	LOCAL CONST Robtarget Tr_meulage_bavure_P130 :=[[66.91934375,115.7860078125,16],[0.0375790299429137,-0.0384114691049443,-0.713777108740491,0.698308395043204],[0,0,0,0],[8.999999E+09,8.999999E+09,8.999999E+09,8.999999E+09,8.999999E+09,8.999999E+09]];
	LOCAL CONST Robtarget Tr_meulage_bavure_P131 :=[[72.78634375,115.0686953125,16],[0.040217072512141,-0.0409917261667762,-0.712641457174476,0.699174097761538],[0,0,0,0],[8.999999E+09,8.999999E+09,8.999999E+09,8.999999E+09,8.999999E+09,8.999999E+09]];
	LOCAL CONST Robtarget Tr_meulage_bavure_P132 :=[[73.607359375,114.957515625,16],[0.0430704475740681,-0.0437750469990952,-0.711474851088136,0.700023012532524],[0,0,0,0],[8.999999E+09,8.999999E+09,8.999999E+09,8.999999E+09,8.999999E+09,8.999999E+09]];
	LOCAL CONST Robtarget Tr_meulage_bavure_P133 :=[[80.8797578125,113.9724765625,16],[0.0463242339768427,-0.0469486652254147,-0.710274730272182,0.70082786454078],[0,0,0,0],[8.999999E+09,8.999999E+09,8.999999E+09,8.999999E+09,8.999999E+09,8.999999E+09]];
	LOCAL CONST Robtarget Tr_meulage_bavure_P134 :=[[81.893921875,113.8622109375,16],[0.0500455236008215,-0.0505782090053766,-0.70903845529879,0.701570922465316],[0,0,0,0],[8.999999E+09,8.999999E+09,8.999999E+09,8.999999E+09,8.999999E+09,8.999999E+09]];
	LOCAL CONST Robtarget Tr_meulage_bavure_P135 :=[[86.0903046875,113.1481953125,16],[0.0541087782813907,-0.0545356720476456,-0.70778179785277,0.702241430859436],[0,0,0,0],[8.999999E+09,8.999999E+09,8.999999E+09,8.999999E+09,8.999999E+09,8.999999E+09]];
	LOCAL CONST Robtarget Tr_meulage_bavure_P136 :=[[87.9428125,112.849546875,16],[0.0582007586477647,-0.0585060712323081,-0.706535976535859,0.70284893482334],[0,0,0,0],[8.999999E+09,8.999999E+09,8.999999E+09,8.999999E+09,8.999999E+09,8.999999E+09]];
	LOCAL CONST Robtarget Tr_meulage_bavure_P137 :=[[89.760375,112.5874921875,16],[0.0619449334526603,-0.0621148803561433,-0.705345034592479,0.703415203868684],[0,0,0,0],[8.999999E+09,8.999999E+09,8.999999E+09,8.999999E+09,8.999999E+09,8.999999E+09]];
	LOCAL CONST Robtarget Tr_meulage_bavure_P138 :=[[96.0940234375,111.0590546875,16],[0.0650697780701425,-0.065095955864691,-0.704246851452174,0.703963644467287],[0,0,0,0],[8.999999E+09,8.999999E+09,8.999999E+09,8.999999E+09,8.999999E+09,8.999999E+09]];
	LOCAL CONST Robtarget Tr_meulage_bavure_P139 :=[[96.4307578125,110.9958203125,16],[0.0675357884502958,-0.0674170712414185,-0.703260439151439,0.704498836413625],[0,0,0,0],[8.999999E+09,8.999999E+09,8.999999E+09,8.999999E+09,8.999999E+09,8.999999E+09]];
	LOCAL CONST Robtarget Tr_meulage_bavure_P140 :=[[106.677734375,109.285953125,16],[0.0695409234803893,-0.0692837834926727,-0.702387001473537,0.704993842148603],[0,0,0,0],[8.999999E+09,8.999999E+09,8.999999E+09,8.999999E+09,8.999999E+09,8.999999E+09]];
	LOCAL CONST Robtarget Tr_meulage_bavure_P141 :=[[106.9891640625,109.2307109375,16],[0.0713921073001013,-0.0710053649896085,-0.70159983106773,0.705421209068508],[0,0,0,0],[8.999999E+09,8.999999E+09,8.999999E+09,8.999999E+09,8.999999E+09,8.999999E+09]];
	LOCAL CONST Robtarget Tr_meulage_bavure_P142 :=[[107.1989453125,109.1865234375,16],[0.0732993553122748,-0.0727933096486914,-0.700883234161866,0.705755645143557],[0,0,0,0],[8.999999E+09,8.999999E+09,8.999999E+09,8.999999E+09,8.999999E+09,8.999999E+09]];
	LOCAL CONST Robtarget Tr_meulage_bavure_P143 :=[[110.56125,108.47396875,16],[0.0752309363699142,-0.0746187293208283,-0.700247555166698,0.705992714502433],[0,0,0,0],[8.999999E+09,8.999999E+09,8.999999E+09,8.999999E+09,8.999999E+09,8.999999E+09]];
	LOCAL CONST Robtarget Tr_meulage_bavure_P144 :=[[111.3198828125,108.289640625,16],[0.0769389781355609,-0.076236764322119,-0.699716860698982,0.706161924959644],[0,0,0,0],[8.999999E+09,8.999999E+09,8.999999E+09,8.999999E+09,8.999999E+09,8.999999E+09]];
	LOCAL CONST Robtarget Tr_meulage_bavure_P145 :=[[112.3602265625,108.048890625,16],[0.0781115130178079,-0.0773402560327233,-0.699326258671287,0.706300120532116],[0,0,0,0],[8.999999E+09,8.999999E+09,8.999999E+09,8.999999E+09,8.999999E+09,8.999999E+09]];
	LOCAL CONST Robtarget Tr_meulage_bavure_P146 :=[[114.5588359375,107.543515625,16],[0.0785747149746875,-0.0777587433548293,-0.699095336504751,0.706431385539907],[0,0,0,0],[8.999999E+09,8.999999E+09,8.999999E+09,8.999999E+09,8.999999E+09,8.999999E+09]];
	LOCAL CONST Robtarget Tr_meulage_bavure_P147 :=[[115.668765625,107.266140625,16],[0.0784214795360947,-0.0775843590394273,-0.699009918050557,0.706552102287415],[0,0,0,0],[8.999999E+09,8.999999E+09,8.999999E+09,8.999999E+09,8.999999E+09,8.999999E+09]];
	LOCAL CONST Robtarget Tr_meulage_bavure_P148 :=[[117.5694609375,106.84359375,16],[0.0780069203121761,-0.0771676079432631,-0.699025386011006,0.706628325486524],[0,0,0,0],[8.999999E+09,8.999999E+09,8.999999E+09,8.999999E+09,8.999999E+09,8.999999E+09]];
	LOCAL CONST Robtarget Tr_meulage_bavure_P149 :=[[118.382015625,106.655640625,16],[0.0777860523380435,-0.0769565613223954,-0.699083246410587,0.706618448895251],[0,0,0,0],[8.999999E+09,8.999999E+09,8.999999E+09,8.999999E+09,8.999999E+09,8.999999E+09]];
	LOCAL CONST Robtarget Tr_meulage_bavure_P150 :=[[121.6917734375,105.9990546875,16],[0.0781312083527598,-0.077318092245178,-0.699136115354537,0.706488583842563],[0,0,0,0],[8.999999E+09,8.999999E+09,8.999999E+09,8.999999E+09,8.999999E+09,8.999999E+09]];
	LOCAL CONST Robtarget Tr_meulage_bavure_P151 :=[[125.2111171875,105.2392265625,16],[0.0792169084017852,-0.078423438108987,-0.699154110679908,0.706227991018351],[0,0,0,0],[8.999999E+09,8.999999E+09,8.999999E+09,8.999999E+09,8.999999E+09,8.999999E+09]];
	LOCAL CONST Robtarget Tr_meulage_bavure_P152 :=[[126.6580234375,104.8870234375,16],[0.0809905250458525,-0.0802193534282553,-0.699128968723034,0.705849895714816],[0,0,0,0],[8.999999E+09,8.999999E+09,8.999999E+09,8.999999E+09,8.999999E+09,8.999999E+09]];
	LOCAL CONST Robtarget Tr_meulage_bavure_P153 :=[[129.6603984375,104.143984375,16],[0.0832551345128652,-0.0825101821253249,-0.699069483083656,0.705381109928555],[0,0,0,0],[8.999999E+09,8.999999E+09,8.999999E+09,8.999999E+09,8.999999E+09,8.999999E+09]];
	LOCAL CONST Robtarget Tr_meulage_bavure_P154 :=[[136.354125,102.4169609375,16],[0.0857848622766101,-0.0850709210273251,-0.698988120213109,0.70485424280534],[0,0,0,0],[8.999999E+09,8.999999E+09,8.999999E+09,8.999999E+09,8.999999E+09,8.999999E+09]];
	LOCAL CONST Robtarget Tr_meulage_bavure_P155 :=[[137.42846875,102.1511875,16],[0.0884091672402083,-0.0877319052022491,-0.698897826468415,0.704293092480114],[0,0,0,0],[8.999999E+09,8.999999E+09,8.999999E+09,8.999999E+09,8.999999E+09,8.999999E+09]];
	LOCAL CONST Robtarget Tr_meulage_bavure_P156 :=[[144.5833125,100.26434375,16],[0.0910431915599839,-0.0904067032944326,-0.698798168569051,0.703717901487908],[0,0,0,0],[8.999999E+09,8.999999E+09,8.999999E+09,8.999999E+09,8.999999E+09,8.999999E+09]];
	LOCAL CONST Robtarget Tr_meulage_bavure_P157 :=[[146.926640625,99.6148046875,16],[0.0936691483507536,-0.0930756350342028,-0.698683585512406,0.703138865478046],[0,0,0,0],[8.999999E+09,8.999999E+09,8.999999E+09,8.999999E+09,8.999999E+09,8.999999E+09]];
	LOCAL CONST Robtarget Tr_meulage_bavure_P158 :=[[150.95953125,98.4415625,16],[0.0962879304034066,-0.0957394224747977,-0.69855392139274,0.702556059222072],[0,0,0,0],[8.999999E+09,8.999999E+09,8.999999E+09,8.999999E+09,8.999999E+09,8.999999E+09]];
	LOCAL CONST Robtarget Tr_meulage_bavure_P159 :=[[153.138734375,97.7918125,16],[0.0988916895437435,-0.0983883422839826,-0.698404120332552,0.701977102578359],[0,0,0,0],[8.999999E+09,8.999999E+09,8.999999E+09,8.999999E+09,8.999999E+09,8.999999E+09]];
	LOCAL CONST Robtarget Tr_meulage_bavure_P160 :=[[157.757078125,96.4455546875,16],[0.101440612933847,-0.100981536227335,-0.698236939472659,0.701411225847311],[0,0,0,0],[8.999999E+09,8.999999E+09,8.999999E+09,8.999999E+09,8.999999E+09,8.999999E+09]];
	LOCAL CONST Robtarget Tr_meulage_bavure_P161 :=[[158.63409375,96.21628125,16],[0.103869656310797,-0.103455017724827,-0.698066701122684,0.70086449088902],[0,0,0,0],[8.999999E+09,8.999999E+09,8.999999E+09,8.999999E+09,8.999999E+09,8.999999E+09]];
	LOCAL CONST Robtarget Tr_meulage_bavure_P162 :=[[161.731328125,95.3334375,16],[0.106127055185058,-0.105757019641076,-0.697903326027202,0.700345235205147],[0,0,0,0],[8.999999E+09,8.999999E+09,8.999999E+09,8.999999E+09,8.999999E+09,8.999999E+09]];
	LOCAL CONST Robtarget Tr_meulage_bavure_P163 :=[[163.41271875,94.773984375,16],[0.108205069351474,-0.107879192972837,-0.697749227537857,0.699856955499119],[0,0,0,0],[8.999999E+09,8.999999E+09,8.999999E+09,8.999999E+09,8.999999E+09,8.999999E+09]];
	LOCAL CONST Robtarget Tr_meulage_bavure_P164 :=[[168.711796875,93.117984375,16],[0.110163902620429,-0.109882603679943,-0.697601214294859,0.699387070070852],[0,0,0,0],[8.999999E+09,8.999999E+09,8.999999E+09,8.999999E+09,8.999999E+09,8.999999E+09]];
	LOCAL CONST Robtarget Tr_meulage_bavure_P165 :=[[169.002984375,93.037046875,16],[0.112115837692814,-0.11188027121235,-0.697446164040501,0.698914652956339],[0,0,0,0],[8.999999E+09,8.999999E+09,8.999999E+09,8.999999E+09,8.999999E+09,8.999999E+09]];
	LOCAL CONST Robtarget Tr_meulage_bavure_P166 :=[[175.044734375,91.0927421875,16],[0.114161085801191,-0.113974890865321,-0.697275818516395,0.698414922272729],[0,0,0,0],[8.999999E+09,8.999999E+09,8.999999E+09,8.999999E+09,8.999999E+09,8.999999E+09]];
	LOCAL CONST Robtarget Tr_meulage_bavure_P167 :=[[175.713875,90.8525703125,16],[0.116327655332839,-0.116195967636685,-0.697088341701476,0.697878368753198],[0,0,0,0],[8.999999E+09,8.999999E+09,8.999999E+09,8.999999E+09,8.999999E+09,8.999999E+09]];
	LOCAL CONST Robtarget Tr_meulage_bavure_P168 :=[[177.1794375,90.3878515625,16],[0.118529478570234,-0.118459490986501,-0.696901735552245,0.697313475195594],[0,0,0,0],[8.999999E+09,8.999999E+09,8.999999E+09,8.999999E+09,8.999999E+09,8.999999E+09]];
	LOCAL CONST Robtarget Tr_meulage_bavure_P169 :=[[180.194765625,89.338625,16],[0.120588784077744,-0.120590468458572,-0.696753129059677,0.69674339696702],[0,0,0,0],[8.999999E+09,8.999999E+09,8.999999E+09,8.999999E+09,8.999999E+09,8.999999E+09]];
	LOCAL CONST Robtarget Tr_meulage_bavure_P170 :=[[182.01146875,88.6708671875,16],[0.122306368602409,-0.122391776429605,-0.696684495612379,0.696198332973458],[0,0,0,0],[8.999999E+09,8.999999E+09,8.999999E+09,8.999999E+09,8.999999E+09,8.999999E+09]];
	LOCAL CONST Robtarget Tr_meulage_bavure_P171 :=[[185.929625,87.2135,16],[0.123567193506988,-0.123751009683332,-0.696727295823529,0.695692397217042],[0,0,0,0],[8.999999E+09,8.999999E+09,8.999999E+09,8.999999E+09,8.999999E+09,8.999999E+09]];
	LOCAL CONST Robtarget Tr_meulage_bavure_P172 :=[[187.18065625,86.7315078125,16],[0.124415620474812,-0.124713739181367,-0.696880996836631,0.695215155825341],[0,0,0,0],[8.999999E+09,8.999999E+09,8.999999E+09,8.999999E+09,8.999999E+09,8.999999E+09]];
	LOCAL CONST Robtarget Tr_meulage_bavure_P173 :=[[189.04584375,86.04696875,16],[0.125074969784971,-0.125504974941815,-0.697111566398052,0.69472312268428],[0,0,0,0],[8.999999E+09,8.999999E+09,8.999999E+09,8.999999E+09,8.999999E+09,8.999999E+09]];
	LOCAL CONST Robtarget Tr_meulage_bavure_P174 :=[[190.664125,85.3816796875,16],[0.125898358033854,-0.126480701100316,-0.697359329420033,0.694148544163563],[0,0,0,0],[8.999999E+09,8.999999E+09,8.999999E+09,8.999999E+09,8.999999E+09,8.999999E+09]];
	LOCAL CONST Robtarget Tr_meulage_bavure_P175 :=[[192.474609375,84.74475,16],[0.127251837277854,-0.128012368352486,-0.697561606568862,0.693417340783504],[0,0,0,0],[8.999999E+09,8.999999E+09,8.999999E+09,8.999999E+09,8.999999E+09,8.999999E+09]];
	LOCAL CONST Robtarget Tr_meulage_bavure_P176 :=[[194.93378125,83.8551015625,16],[0.129383618966927,-0.130354980774212,-0.697672769672953,0.692473945060207],[0,0,0,0],[8.999999E+09,8.999999E+09,8.999999E+09,8.999999E+09,8.999999E+09,8.999999E+09]];
	LOCAL CONST Robtarget Tr_meulage_bavure_P177 :=[[196.478875,83.225859375,16],[0.132323925738124,-0.133543900842516,-0.697677993470186,0.691304435579891],[0,0,0,0],[8.999999E+09,8.999999E+09,8.999999E+09,8.999999E+09,8.999999E+09,8.999999E+09]];
	LOCAL CONST Robtarget Tr_meulage_bavure_P178 :=[[200.12365625,81.8095390625,16],[0.135877207452713,-0.137388271043078,-0.697605868715162,0.689933257213197],[0,0,0,0],[8.999999E+09,8.999999E+09,8.999999E+09,8.999999E+09,8.999999E+09,8.999999E+09]];
	LOCAL CONST Robtarget Tr_meulage_bavure_P179 :=[[202.561578125,80.75653125,16],[0.139685278222459,-0.141531070512551,-0.697518656155899,0.688421893494065],[0,0,0,0],[8.999999E+09,8.999999E+09,8.999999E+09,8.999999E+09,8.999999E+09,8.999999E+09]];
	LOCAL CONST Robtarget Tr_meulage_bavure_P180 :=[[207.698796875,78.43090625,16],[0.143350747480375,-0.145574635078128,-0.697498867206909,0.686843445818453],[0,0,0,0],[8.999999E+09,8.999999E+09,8.999999E+09,8.999999E+09,8.999999E+09,8.999999E+09]];
	LOCAL CONST Robtarget Tr_meulage_bavure_P181 :=[[209.555171875,77.6030546875,16],[0.146540725641296,-0.149180855171853,-0.697618889464421,0.685272772873069],[0,0,0,0],[8.999999E+09,8.999999E+09,8.999999E+09,8.999999E+09,8.999999E+09,8.999999E+09]];
	LOCAL CONST Robtarget Tr_meulage_bavure_P182 :=[[210.891359375,77.0095234375,16],[0.149040228183799,-0.152126413175283,-0.697928299674523,0.68376944455772],[0,0,0,0],[8.999999E+09,8.999999E+09,8.999999E+09,8.999999E+09,8.999999E+09,8.999999E+09]];
	LOCAL CONST Robtarget Tr_meulage_bavure_P183 :=[[212.986875,76.031890625,16],[0.150734443360395,-0.154289349959885,-0.698460976711582,0.682368073758504],[0,0,0,0],[8.999999E+09,8.999999E+09,8.999999E+09,8.999999E+09,8.999999E+09,8.999999E+09]];
	LOCAL CONST Robtarget Tr_meulage_bavure_P184 :=[[217.078546875,74.016234375,16],[0.151570317945741,-0.155607772630321,-0.699233612155391,0.681091047839407],[0,0,0,0],[8.999999E+09,8.999999E+09,8.999999E+09,8.999999E+09,8.999999E+09,8.999999E+09]];
	LOCAL CONST Robtarget Tr_meulage_bavure_P185 :=[[218.941953125,73.112125,16],[0.151569402372408,-0.156092119138138,-0.700237370211066,0.679948227416857],[0,0,0,0],[8.999999E+09,8.999999E+09,8.999999E+09,8.999999E+09,8.999999E+09,8.999999E+09]];
	LOCAL CONST Robtarget Tr_meulage_bavure_P186 :=[[219.0621875,73.06121875,16],[0.150837702259073,-0.155840185661068,-0.701442332980961,0.678925973588103],[0,0,0,0],[8.999999E+09,8.999999E+09,8.999999E+09,8.999999E+09,8.999999E+09,8.999999E+09]];
	LOCAL CONST Robtarget Tr_meulage_bavure_P187 :=[[219.1090625,73.033109375,16],[0.149636648993526,-0.155109844533247,-0.702776618858019,0.677978490361863],[0,0,0,0],[8.999999E+09,8.999999E+09,8.999999E+09,8.999999E+09,8.999999E+09,8.999999E+09]];
	LOCAL CONST Robtarget Tr_meulage_bavure_P188 :=[[222.09015625,71.6129140625,16],[0.148574336094181,-0.154522304802513,-0.704087568238217,0.676985391441416],[0,0,0,0],[8.999999E+09,8.999999E+09,8.999999E+09,8.999999E+09,8.999999E+09,8.999999E+09]];
	LOCAL CONST Robtarget Tr_meulage_bavure_P189 :=[[229.641546875,68.055234375,16],[0.148626996287793,-0.155089341077337,-0.705134905379677,0.675752970747344],[0,0,0,0],[8.999999E+09,8.999999E+09,8.999999E+09,8.999999E+09,8.999999E+09,8.999999E+09]];
	LOCAL CONST Robtarget Tr_meulage_bavure_P190 :=[[230.11071875,67.8279140625,16],[0.151271074807113,-0.158361042480802,-0.705554971353023,0.673966634597091],[0,0,0,0],[8.999999E+09,8.999999E+09,8.999999E+09,8.999999E+09,8.999999E+09,8.999999E+09]];
	LOCAL CONST Robtarget Tr_meulage_bavure_P191 :=[[233.1743125,66.54559375,16],[0.158480102126182,-0.166430569449805,-0.704809140639182,0.671140073348438],[0,0,0,0],[8.999999E+09,8.999999E+09,8.999999E+09,8.999999E+09,8.999999E+09,8.999999E+09]];
	LOCAL CONST Robtarget Tr_meulage_bavure_P192 :=[[233.944765625,66.22134375,16],[0.172471661081484,-0.181663624911472,-0.702094674614285,0.666569517294393],[0,0,0,0],[8.999999E+09,8.999999E+09,8.999999E+09,8.999999E+09,8.999999E+09,8.999999E+09]];
	LOCAL CONST Robtarget Tr_meulage_bavure_P193 :=[[234.4685,65.9126875,16],[0.195272456379888,-0.206245163845634,-0.696254711205549,0.659212391641518],[0,0,0,0],[8.999999E+09,8.999999E+09,8.999999E+09,8.999999E+09,8.999999E+09,8.999999E+09]];
	LOCAL CONST Robtarget Tr_meulage_bavure_P194 :=[[235.857546875,65.32159375,16],[0.227792969698998,-0.24119253559603,-0.685838349962404,0.647736274612836],[0,0,0,0],[8.999999E+09,8.999999E+09,8.999999E+09,8.999999E+09,8.999999E+09,8.999999E+09]];
	LOCAL CONST Robtarget Tr_meulage_bavure_P195 :=[[237.085015625,64.44748046875,16],[0.268887533298227,-0.285326947579369,-0.669496083625712,0.63092235768886],[0,0,0,0],[8.999999E+09,8.999999E+09,8.999999E+09,8.999999E+09,8.999999E+09,8.999999E+09]];
	LOCAL CONST Robtarget Tr_meulage_bavure_P196 :=[[237.9425625,63.1903984375,16],[0.314996141790336,-0.334870453464709,-0.646850326102626,0.608460241654678],[0,0,0,0],[8.999999E+09,8.999999E+09,8.999999E+09,8.999999E+09,8.999999E+09,8.999999E+09]];
	LOCAL CONST Robtarget Tr_meulage_bavure_P197 :=[[238.0418125,63.07073828125,16],[0.361424808772667,-0.384786321985673,-0.619044160812946,0.581460162848475],[0,0,0,0],[8.999999E+09,8.999999E+09,8.999999E+09,8.999999E+09,8.999999E+09,8.999999E+09]];
	LOCAL CONST Robtarget Tr_meulage_bavure_P198 :=[[238.087640625,62.9619765625,16],[0.404605659191079,-0.431207701831069,-0.588094753981249,0.551814043652256],[0,0,0,0],[8.999999E+09,8.999999E+09,8.999999E+09,8.999999E+09,8.999999E+09,8.999999E+09]];
	LOCAL CONST Robtarget Tr_meulage_bavure_P199 :=[[238.506046875,60.62127734375,16],[0.443062387855305,-0.472484667298788,-0.555752974041069,0.521145460960772],[0,0,0,0],[8.999999E+09,8.999999E+09,8.999999E+09,8.999999E+09,8.999999E+09,8.999999E+09]];
	LOCAL CONST Robtarget Tr_meulage_bavure_P200 :=[[238.6093125,59.7001328125,16],[0.476650321376658,-0.508389052787827,-0.52319014626542,0.490527382505598],[0,0,0,0],[8.999999E+09,8.999999E+09,8.999999E+09,8.999999E+09,8.999999E+09,8.999999E+09]];
	LOCAL CONST Robtarget Tr_meulage_bavure_P201 :=[[237.7109375,57.469390625,16],[0.505451156136112,-0.53895486429405,-0.491501652997141,0.460947836653485],[0,0,0,0],[8.999999E+09,8.999999E+09,8.999999E+09,8.999999E+09,8.999999E+09,8.999999E+09]];
	LOCAL CONST Robtarget Tr_meulage_bavure_P202 :=[[236.879703125,55.57473828125,16],[0.529331236729187,-0.564002254730795,-0.462148127760641,0.433738407901194],[0,0,0,0],[8.999999E+09,8.999999E+09,8.999999E+09,8.999999E+09,8.999999E+09,8.999999E+09]];
	LOCAL CONST Robtarget Tr_meulage_bavure_P203 :=[[236.66284375,55.11083984375,16],[0.548233372494373,-0.583447016687868,-0.436664316627856,0.410309666697484],[0,0,0,0],[8.999999E+09,8.999999E+09,8.999999E+09,8.999999E+09,8.999999E+09,8.999999E+09]];
	LOCAL CONST Robtarget Tr_meulage_bavure_P204 :=[[235.0753125,52.03003125,16],[0.562452491386192,-0.597603777768636,-0.416104904645074,0.391629452493596],[0,0,0,0],[8.999999E+09,8.999999E+09,8.999999E+09,8.999999E+09,8.999999E+09,8.999999E+09]];
	LOCAL CONST Robtarget Tr_meulage_bavure_P205 :=[[232.848875,47.99112109375,16],[0.572670247409118,-0.607197499281822,-0.400686686586718,0.377902320435371],[0,0,0,0],[8.999999E+09,8.999999E+09,8.999999E+09,8.999999E+09,8.999999E+09,8.999999E+09]];
	LOCAL CONST Robtarget Tr_meulage_bavure_P206 :=[[231.788703125,45.97287109375,16],[0.579797402910104,-0.613235537289396,-0.3898050973045,0.368550042056046],[0,0,0,0],[8.999999E+09,8.999999E+09,8.999999E+09,8.999999E+09,8.999999E+09,8.999999E+09]];
	LOCAL CONST Robtarget Tr_meulage_bavure_P207 :=[[231.750421875,46.01022265625,16],[0.584743800948948,-0.616698687680699,-0.382440881141462,0.362624307371171],[0,0,0,0],[8.999999E+09,8.999999E+09,8.999999E+09,8.999999E+09,8.999999E+09,8.999999E+09]];
	LOCAL CONST Robtarget Tr_meulage_bavure_P208 :=[[230.563046875,43.4813828125,16],[0.588303582827908,-0.618443461707875,-0.377476158934893,0.359079835883867],[0,0,0,0],[8.999999E+09,8.999999E+09,8.999999E+09,8.999999E+09,8.999999E+09,8.999999E+09]];
	LOCAL CONST Robtarget Tr_meulage_bavure_P209 :=[[228.135625,38.742125,16],[0.591075423099639,-0.619138479944678,-0.373956669203322,0.357006717608694],[0,0,0,0],[8.999999E+09,8.999999E+09,8.999999E+09,8.999999E+09,8.999999E+09,8.999999E+09]];
	LOCAL CONST Robtarget Tr_meulage_bavure_P210 :=[[227.6539375,37.97744921875,16],[0.59346983022117,-0.619233588321481,-0.371194119980086,0.355750262127757],[0,0,0,0],[8.999999E+09,8.999999E+09,8.999999E+09,8.999999E+09,8.999999E+09,8.999999E+09]];
	LOCAL CONST Robtarget Tr_meulage_bavure_P211 :=[[227.583375,37.84625390625,16],[0.59578771747521,-0.619083199083303,-0.368651892343638,0.354779890340359],[0,0,0,0],[8.999999E+09,8.999999E+09,8.999999E+09,8.999999E+09,8.999999E+09,8.999999E+09]];
	LOCAL CONST Robtarget Tr_meulage_bavure_P212 :=[[223.232234375,29.75045703125,16],[0.59826322315855,-0.618948699501958,-0.365912211100707,0.353683300380678],[0,0,0,0],[8.999999E+09,8.999999E+09,8.999999E+09,8.999999E+09,8.999999E+09,8.999999E+09]];
	LOCAL CONST Robtarget Tr_meulage_bavure_P213 :=[[222.742609375,28.879546875,16],[0.601110196290616,-0.619074471589474,-0.362582673927974,0.35206126612979],[0,0,0,0],[8.999999E+09,8.999999E+09,8.999999E+09,8.999999E+09,8.999999E+09,8.999999E+09]];
	LOCAL CONST Robtarget Tr_meulage_bavure_P214 :=[[219.652765625,22.688568359375,16],[0.604470518421326,-0.619625642008761,-0.358389216634608,0.349623548298331],[0,0,0,0],[8.999999E+09,8.999999E+09,8.999999E+09,8.999999E+09,8.999999E+09,8.999999E+09]];
	LOCAL CONST Robtarget Tr_meulage_bavure_P215 :=[[218.990046875,21.3121328125,16],[0.608276493688391,-0.620552871503657,-0.353416807429074,0.346425173914026],[0,0,0,0],[8.999999E+09,8.999999E+09,8.999999E+09,8.999999E+09,8.999999E+09,8.999999E+09]];
	LOCAL CONST Robtarget Tr_meulage_bavure_P216 :=[[218.1641875,19.516814453125,16],[0.612202390644332,-0.6215539324952,-0.348209714398515,0.342970751941944],[0,0,0,0],[8.999999E+09,8.999999E+09,8.999999E+09,8.999999E+09,8.999999E+09,8.999999E+09]];
	LOCAL CONST Robtarget Tr_meulage_bavure_P217 :=[[215.843265625,15.1568603515625,16],[0.615711006556747,-0.622118377345017,-0.343722099195397,0.340182009370264],[0,0,0,0],[8.999999E+09,8.999999E+09,8.999999E+09,8.999999E+09,8.999999E+09,8.999999E+09]];
	LOCAL CONST Robtarget Tr_meulage_bavure_P218 :=[[215.603765625,14.73193359375,16],[0.618247194410525,-0.621700174240876,-0.34098922432466,0.339095338875138],[0,0,0,0],[8.999999E+09,8.999999E+09,8.999999E+09,8.999999E+09,8.999999E+09,8.999999E+09]];
	LOCAL CONST Robtarget Tr_meulage_bavure_P219 :=[[215.48725,14.5715634765625,16],[0.619428558964651,-0.619963866268426,-0.340700330946559,0.340406153518684],[0,0,0,0],[8.999999E+09,8.999999E+09,8.999999E+09,8.999999E+09,8.999999E+09,8.999999E+09]];
	LOCAL CONST Robtarget Tr_meulage_bavure_P220 :=[[212.94371875,10.92562890625,16],[0.619189685973086,-0.616882730457898,-0.34291302665433,0.34419541803767],[0,0,0,0],[8.999999E+09,8.999999E+09,8.999999E+09,8.999999E+09,8.999999E+09,8.999999E+09]];
	LOCAL CONST Robtarget Tr_meulage_bavure_P221 :=[[210.711859375,7.6824033203125,16],[0.617793467753272,-0.612757654465243,-0.347038617328745,0.349890677466824],[0,0,0,0],[8.999999E+09,8.999999E+09,8.999999E+09,8.999999E+09,8.999999E+09,8.999999E+09]];
	LOCAL CONST Robtarget Tr_meulage_bavure_P222 :=[[209.336421875,5.25592041015625,16],[0.615729233509894,-0.608088125169878,-0.352115617639173,0.356540228926954],[0,0,0,0],[8.999999E+09,8.999999E+09,8.999999E+09,8.999999E+09,8.999999E+09,8.999999E+09]];
	LOCAL CONST Robtarget Tr_meulage_bavure_P223 :=[[208.604984375,3.98187255859375,16],[0.613532173472829,-0.603419982946631,-0.357177068427192,0.363162688177283],[0,0,0,0],[8.999999E+09,8.999999E+09,8.999999E+09,8.999999E+09,8.999999E+09,8.999999E+09]];
	LOCAL CONST Robtarget Tr_meulage_bavure_P224 :=[[206.372984375,-0.804412841796875,16],[0.611662197159133,-0.59922168111387,-0.361469981964712,0.368974505336019],[0,0,0,0],[8.999999E+09,8.999999E+09,8.999999E+09,8.999999E+09,8.999999E+09,8.999999E+09]];
	LOCAL CONST Robtarget Tr_meulage_bavure_P225 :=[[205.655703125,-2.33804321289063,16],[0.610428440285061,-0.595774575282164,-0.364562330984876,0.373529224513126],[0,0,0,0],[8.999999E+09,8.999999E+09,8.999999E+09,8.999999E+09,8.999999E+09,8.999999E+09]];
	LOCAL CONST Robtarget Tr_meulage_bavure_P226 :=[[205.306515625,-3.13638305664063,16],[0.609970630238294,-0.593221869097205,-0.366292565633338,0.376634306235191],[0,0,0,0],[8.999999E+09,8.999999E+09,8.999999E+09,8.999999E+09,8.999999E+09,8.999999E+09]];
	LOCAL CONST Robtarget Tr_meulage_bavure_P227 :=[[203.0261875,-7.57730078125,16],[0.610287493058713,-0.591562424509279,-0.366711703652052,0.378319441913082],[0,0,0,0],[8.999999E+09,8.999999E+09,8.999999E+09,8.999999E+09,8.999999E+09,8.999999E+09]];
	LOCAL CONST Robtarget Tr_meulage_bavure_P228 :=[[201.42346875,-10.699615234375,16],[0.611273752937712,-0.590676043388691,-0.366019028972191,0.378782630497203],[0,0,0,0],[8.999999E+09,8.999999E+09,8.999999E+09,8.999999E+09,8.999999E+09,8.999999E+09]];
	LOCAL CONST Robtarget Tr_meulage_bavure_P229 :=[[197.501828125,-18.230896484375,16],[0.612750021112551,-0.59039743156596,-0.364498085131601,0.378298070788474],[0,0,0,0],[8.999999E+09,8.999999E+09,8.999999E+09,8.999999E+09,8.999999E+09,8.999999E+09]];
	LOCAL CONST Robtarget Tr_meulage_bavure_P230 :=[[196.443484375,-20.251861328125,16],[0.614519592787454,-0.590532121989523,-0.362455427247399,0.377178401075405],[0,0,0,0],[8.999999E+09,8.999999E+09,8.999999E+09,8.999999E+09,8.999999E+09,8.999999E+09]];
	LOCAL CONST Robtarget Tr_meulage_bavure_P231 :=[[195.890625,-21.320525390625,16],[0.616387866924389,-0.590909198060636,-0.36018303811425,0.375713316520091],[0,0,0,0],[8.999999E+09,8.999999E+09,8.999999E+09,8.999999E+09,8.999999E+09,8.999999E+09]];
	LOCAL CONST Robtarget Tr_meulage_bavure_P232 :=[[192.78528125,-26.824158203125,16],[0.618192759727046,-0.591385952223848,-0.357926574441675,0.374150951678328],[0,0,0,0],[8.999999E+09,8.999999E+09,8.999999E+09,8.999999E+09,8.999999E+09,8.999999E+09]];
	LOCAL CONST Robtarget Tr_meulage_bavure_P233 :=[[191.961296875,-28.487701171875,16],[0.619788398563889,-0.59181878102234,-0.355918672819268,0.372739546833191],[0,0,0,0],[8.999999E+09,8.999999E+09,8.999999E+09,8.999999E+09,8.999999E+09,8.999999E+09]];
	LOCAL CONST Robtarget Tr_meulage_bavure_P234 :=[[191.71503125,-29.23452734375,16],[0.621010587314961,-0.592072467915302,-0.354413234717379,0.371735527272516],[0,0,0,0],[8.999999E+09,8.999999E+09,8.999999E+09,8.999999E+09,8.999999E+09,8.999999E+09]];
	LOCAL CONST Robtarget Tr_meulage_bavure_P235 :=[[191.2190625,-30.219666015625,16],[0.621717150920934,-0.592020916672666,-0.353636981800015,0.371375690610181],[0,0,0,0],[8.999999E+09,8.999999E+09,8.999999E+09,8.999999E+09,8.999999E+09,8.999999E+09]];
	LOCAL CONST Robtarget Tr_meulage_bavure_P236 :=[[190.413390625,-31.797484375,16],[0.621844618805108,-0.591613368888173,-0.35368880301411,0.371762185325999],[0,0,0,0],[8.999999E+09,8.999999E+09,8.999999E+09,8.999999E+09,8.999999E+09,8.999999E+09]];
	LOCAL CONST Robtarget Tr_meulage_bavure_P237 :=[[189.352296875,-33.64605859375,16],[0.621474786784406,-0.590935626905415,-0.354432305698057,0.372749131350752],[0,0,0,0],[8.999999E+09,8.999999E+09,8.999999E+09,8.999999E+09,8.999999E+09,8.999999E+09]];
	LOCAL CONST Robtarget Tr_meulage_bavure_P238 :=[[188.66540625,-34.951109375,16],[0.620853488883399,-0.590218182218205,-0.35547523483033,0.373926196117189],[0,0,0,0],[8.999999E+09,8.999999E+09,8.999999E+09,8.999999E+09,8.999999E+09,8.999999E+09]];
	LOCAL CONST Robtarget Tr_meulage_bavure_P239 :=[[187.039984375,-37.97381640625,16],[0.620336030294727,-0.589817841504478,-0.356247814205903,0.374680688366368],[0,0,0,0],[8.999999E+09,8.999999E+09,8.999999E+09,8.999999E+09,8.999999E+09,8.999999E+09]];
	LOCAL CONST Robtarget Tr_meulage_bavure_P240 :=[[186.095953125,-39.88458203125,16],[0.62027164381349,-0.590046519008715,-0.356213130566664,0.374460143270959],[0,0,0,0],[8.999999E+09,8.999999E+09,8.999999E+09,8.999999E+09,8.999999E+09,8.999999E+09]];
	LOCAL CONST Robtarget Tr_meulage_bavure_P241 :=[[184.659484375,-42.5355234375,16],[0.620848961703628,-0.591075599173121,-0.355073857767026,0.372959459384133],[0,0,0,0],[8.999999E+09,8.999999E+09,8.999999E+09,8.999999E+09,8.999999E+09,8.999999E+09]];
	LOCAL CONST Robtarget Tr_meulage_bavure_P242 :=[[183.497984375,-44.72093359375,16],[0.622007609011476,-0.592853797057783,-0.352903022008749,0.370257162932856],[0,0,0,0],[8.999999E+09,8.999999E+09,8.999999E+09,8.999999E+09,8.999999E+09,8.999999E+09]];
	LOCAL CONST Robtarget Tr_meulage_bavure_P243 :=[[182.948,-45.741546875,16],[0.623470604116682,-0.595107437368185,-0.350120143436793,0.366807073202319],[0,0,0,0],[8.999999E+09,8.999999E+09,8.999999E+09,8.999999E+09,8.999999E+09,8.999999E+09]];
	LOCAL CONST Robtarget Tr_meulage_bavure_P244 :=[[182.502265625,-46.5653671875,16],[0.624830473684378,-0.59744409125455,-0.347369716800421,0.363292880236285],[0,0,0,0],[8.999999E+09,8.999999E+09,8.999999E+09,8.999999E+09,8.999999E+09,8.999999E+09]];
	LOCAL CONST Robtarget Tr_meulage_bavure_P245 :=[[180.579765625,-49.96437109375,16],[0.625689222370143,-0.599454185968829,-0.345326866083021,0.360440052568486],[0,0,0,0],[8.999999E+09,8.999999E+09,8.999999E+09,8.999999E+09,8.999999E+09,8.999999E+09]];
	LOCAL CONST Robtarget Tr_meulage_bavure_P246 :=[[178.879265625,-52.42295703125,16],[0.625787535266007,-0.600881790469465,-0.344450124057943,0.358727120001225],[0,0,0,0],[8.999999E+09,8.999999E+09,8.999999E+09,8.999999E+09,8.999999E+09,8.999999E+09]];
	LOCAL CONST Robtarget Tr_meulage_bavure_P247 :=[[177.75403125,-54.22612109375,16],[0.625096640484182,-0.601683573776541,-0.344817130388136,0.358234858289601],[0,0,0,0],[8.999999E+09,8.999999E+09,8.999999E+09,8.999999E+09,8.999999E+09,8.999999E+09]];
	LOCAL CONST Robtarget Tr_meulage_bavure_P248 :=[[176.502140625,-56.56321875,16],[0.623836157558886,-0.602041809301397,-0.346081948112199,0.358610364554805],[0,0,0,0],[8.999999E+09,8.999999E+09,8.999999E+09,8.999999E+09,8.999999E+09,8.999999E+09]];
	LOCAL CONST Robtarget Tr_meulage_bavure_P249 :=[[174.892328125,-59.35589453125,16],[0.622391120370798,-0.602317688626201,-0.347602406444529,0.359186946151369],[0,0,0,0],[8.999999E+09,8.999999E+09,8.999999E+09,8.999999E+09,8.999999E+09,8.999999E+09]];
	LOCAL CONST Robtarget Tr_meulage_bavure_P250 :=[[174.53259375,-59.8879375,16],[0.621154712377756,-0.602871615478753,-0.348729548041246,0.359305358802084],[0,0,0,0],[8.999999E+09,8.999999E+09,8.999999E+09,8.999999E+09,8.999999E+09,8.999999E+09]];
	LOCAL CONST Robtarget Tr_meulage_bavure_P251 :=[[172.712578125,-63.39216796875,16],[0.620331837491256,-0.603876425402539,-0.349133232445201,0.358646985544475],[0,0,0,0],[8.999999E+09,8.999999E+09,8.999999E+09,8.999999E+09,8.999999E+09,8.999999E+09]];
	LOCAL CONST Robtarget Tr_meulage_bavure_P252 :=[[171.728453125,-65.503203125,16],[0.619805074760416,-0.605222481505007,-0.349003645355567,0.357412748388586],[0,0,0,0],[8.999999E+09,8.999999E+09,8.999999E+09,8.999999E+09,8.999999E+09,8.999999E+09]];
	LOCAL CONST Robtarget Tr_meulage_bavure_P253 :=[[169.82275,-69.12046875,16],[0.619207693908575,-0.60652948670266,-0.348969562751748,0.35626402826764],[0,0,0,0],[8.999999E+09,8.999999E+09,8.999999E+09,8.999999E+09,8.999999E+09,8.999999E+09]];
	LOCAL CONST Robtarget Tr_meulage_bavure_P254 :=[[168.76715625,-71.4039296875,16],[0.618087663420885,-0.607348493401192,-0.349806991606178,0.355992298390918],[0,0,0,0],[8.999999E+09,8.999999E+09,8.999999E+09,8.999999E+09,8.999999E+09,8.999999E+09]];
	LOCAL CONST Robtarget Tr_meulage_bavure_P255 :=[[167.9378125,-73.0588515625,16],[0.616144959830655,-0.607357422873582,-0.352044103976498,0.357137646028848],[0,0,0,0],[8.999999E+09,8.999999E+09,8.999999E+09,8.999999E+09,8.999999E+09,8.999999E+09]];
	LOCAL CONST Robtarget Tr_meulage_bavure_P256 :=[[166.74378125,-75.276609375,16],[0.613378087222688,-0.606536116562397,-0.355676185075052,0.359688355094935],[0,0,0,0],[8.999999E+09,8.999999E+09,8.999999E+09,8.999999E+09,8.999999E+09,8.999999E+09]];
	LOCAL CONST Robtarget Tr_meulage_bavure_P257 :=[[164.823359375,-78.886203125,16],[0.610086762360184,-0.605171452282996,-0.360170676752647,0.363096046993215],[0,0,0,0],[8.999999E+09,8.999999E+09,8.999999E+09,8.999999E+09,8.999999E+09,8.999999E+09]];
	LOCAL CONST Robtarget Tr_meulage_bavure_P258 :=[[164.210265625,-80.159453125,16],[0.6067464359017,-0.603696402987638,-0.364734016579159,0.366576748704014],[0,0,0,0],[8.999999E+09,8.999999E+09,8.999999E+09,8.999999E+09,8.999999E+09,8.999999E+09]];
	LOCAL CONST Robtarget Tr_meulage_bavure_P259 :=[[159.279296875,-90.4268203125,16],[0.603794572049477,-0.602555269633964,-0.368645944214193,0.369404154841761],[0,0,0,0],[8.999999E+09,8.999999E+09,8.999999E+09,8.999999E+09,8.999999E+09,8.999999E+09]];
	LOCAL CONST Robtarget Tr_meulage_bavure_P260 :=[[159.27728125,-90.43153125,16],[0.601509067955308,-0.602016109948271,-0.371480686790883,0.371167810931474],[0,0,0,0],[8.999999E+09,8.999999E+09,8.999999E+09,8.999999E+09,8.999999E+09,8.999999E+09]];
	LOCAL CONST Robtarget Tr_meulage_bavure_P261 :=[[159.273625,-90.4391953125,16],[0.599964120093679,-0.602129628113578,-0.373150575467244,0.371808571144461],[0,0,0,0],[8.999999E+09,8.999999E+09,8.999999E+09,8.999999E+09,8.999999E+09,8.999999E+09]];
	LOCAL CONST Robtarget Tr_meulage_bavure_P262 :=[[158.607421875,-91.55940625,16],[0.599067473064845,-0.602802801286211,-0.373813700067992,0.371497325856694],[0,0,0,0],[8.999999E+09,8.999999E+09,8.999999E+09,8.999999E+09,8.999999E+09,8.999999E+09]];
	LOCAL CONST Robtarget Tr_meulage_bavure_P263 :=[[157.8125625,-93.275375,16],[0.598655714200807,-0.603859956588914,-0.373739036855634,0.370518044113076],[0,0,0,0],[8.999999E+09,8.999999E+09,8.999999E+09,8.999999E+09,8.999999E+09,8.999999E+09]];
	LOCAL CONST Robtarget Tr_meulage_bavure_P264 :=[[156.013921875,-96.855515625,16],[0.598581633581101,-0.605145309120703,-0.373164557711938,0.369117048720652],[0,0,0,0],[8.999999E+09,8.999999E+09,8.999999E+09,8.999999E+09,8.999999E+09,8.999999E+09]];
	LOCAL CONST Robtarget Tr_meulage_bavure_P265 :=[[154.408453125,-99.789203125,16],[0.598741656024643,-0.606547397296493,-0.372258274988102,0.367467632420327],[0,0,0,0],[8.999999E+09,8.999999E+09,8.999999E+09,8.999999E+09,8.999999E+09,8.999999E+09]];
	LOCAL CONST Robtarget Tr_meulage_bavure_P266 :=[[153.829828125,-100.938015625,16],[0.599111908948481,-0.60801253502702,-0.371071109870387,0.365639042261192],[0,0,0,0],[8.999999E+09,8.999999E+09,8.999999E+09,8.999999E+09,8.999999E+09,8.999999E+09]];
	LOCAL CONST Robtarget Tr_meulage_bavure_P267 :=[[153.0649375,-102.244765625,16],[0.599724034156747,-0.609571192908333,-0.369547441468825,0.363577683769115],[0,0,0,0],[8.999999E+09,8.999999E+09,8.999999E+09,8.999999E+09,8.999999E+09,8.999999E+09]];
	LOCAL CONST Robtarget Tr_meulage_bavure_P268 :=[[150.26190625,-107.945859375,16],[0.600618817736741,-0.611240459447048,-0.367626408072759,0.361238094064016],[0,0,0,0],[8.999999E+09,8.999999E+09,8.999999E+09,8.999999E+09,8.999999E+09,8.999999E+09]];
	LOCAL CONST Robtarget Tr_meulage_bavure_P269 :=[[149.97125,-108.5094296875,16],[0.601781252200874,-0.6130081873259,-0.365324582278095,0.358633847195575],[0,0,0,0],[8.999999E+09,8.999999E+09,8.999999E+09,8.999999E+09,8.999999E+09,8.999999E+09]];
	LOCAL CONST Robtarget Tr_meulage_bavure_P270 :=[[149.841921875,-108.737109375,16],[0.603099595811995,-0.614763102362251,-0.362825686515417,0.355942027175726],[0,0,0,0],[8.999999E+09,8.999999E+09,8.999999E+09,8.999999E+09,8.999999E+09,8.999999E+09]];
	LOCAL CONST Robtarget Tr_meulage_bavure_P271 :=[[148.19159375,-111.5269921875,16],[0.604381813712803,-0.616290646069509,-0.360473121939606,0.353507554628702],[0,0,0,0],[8.999999E+09,8.999999E+09,8.999999E+09,8.999999E+09,8.999999E+09,8.999999E+09]];
	LOCAL CONST Robtarget Tr_meulage_bavure_P272 :=[[147.971859375,-111.859875,16],[0.605406221586117,-0.617363609773654,-0.358664431601985,0.351717650531913],[0,0,0,0],[8.999999E+09,8.999999E+09,8.999999E+09,8.999999E+09,8.999999E+09,8.999999E+09]];
	LOCAL CONST Robtarget Tr_meulage_bavure_P273 :=[[147.5519375,-112.6409296875,16],[0.606016266100963,-0.617826031383224,-0.357686791491451,0.350849596492364],[0,0,0,0],[8.999999E+09,8.999999E+09,8.999999E+09,8.999999E+09,8.999999E+09,8.999999E+09]];
	LOCAL CONST Robtarget Tr_meulage_bavure_P274 :=[[146.0570625,-115.0536171875,16],[0.606201132604477,-0.617685600677894,-0.357557374750242,0.35090940327377],[0,0,0,0],[8.999999E+09,8.999999E+09,8.999999E+09,8.999999E+09,8.999999E+09,8.999999E+09]];
	LOCAL CONST Robtarget Tr_meulage_bavure_P275 :=[[143.955203125,-118.973203125,16],[0.606101570923346,-0.617112593766817,-0.358012611863592,0.35162466080361],[0,0,0,0],[8.999999E+09,8.999999E+09,8.999999E+09,8.999999E+09,8.999999E+09,8.999999E+09]];
	LOCAL CONST Robtarget Tr_meulage_bavure_P276 :=[[143.357421875,-120.373765625,16],[0.6059844558601,-0.616377956599261,-0.358581089829075,0.352534616586018],[0,0,0,0],[8.999999E+09,8.999999E+09,8.999999E+09,8.999999E+09,8.999999E+09,8.999999E+09]];
	LOCAL CONST Robtarget Tr_meulage_bavure_P277 :=[[142.211671875,-123.1184375,16],[0.606111846959739,-0.615785572563122,-0.358782110409862,0.353145798287346],[0,0,0,0],[8.999999E+09,8.999999E+09,8.999999E+09,8.999999E+09,8.999999E+09,8.999999E+09]];
	LOCAL CONST Robtarget Tr_meulage_bavure_P278 :=[[141.69628125,-124.1225625,16],[0.606639211689127,-0.615512883122357,-0.358335319481018,0.353169302692116],[0,0,0,0],[8.999999E+09,8.999999E+09,8.999999E+09,8.999999E+09,8.999999E+09,8.999999E+09]];
	LOCAL CONST Robtarget Tr_meulage_bavure_P279 :=[[141.450984375,-124.770234375,16],[0.607551268446271,-0.615555230777337,-0.357261024378716,0.352615618672595],[0,0,0,0],[8.999999E+09,8.999999E+09,8.999999E+09,8.999999E+09,8.999999E+09,8.999999E+09]];
	LOCAL CONST Robtarget Tr_meulage_bavure_P280 :=[[140.48821875,-126.753109375,16],[0.60860471686433,-0.615722965428547,-0.355948085233736,0.351833041473938],[0,0,0,0],[8.999999E+09,8.999999E+09,8.999999E+09,8.999999E+09,8.999999E+09,8.999999E+09]];
	LOCAL CONST Robtarget Tr_meulage_bavure_P281 :=[[139.2965625,-128.884140625,16],[0.609412114607907,-0.615649493857614,-0.355059221578392,0.351461981520233],[0,0,0,0],[8.999999E+09,8.999999E+09,8.999999E+09,8.999999E+09,8.999999E+09,8.999999E+09]];
	LOCAL CONST Robtarget Tr_meulage_bavure_P282 :=[[138.7163125,-129.7308828125,16],[0.609548490329035,-0.61492304981615,-0.355329209696512,0.352223556110109],[0,0,0,0],[8.999999E+09,8.999999E+09,8.999999E+09,8.999999E+09,8.999999E+09,8.999999E+09]];
	LOCAL CONST Robtarget Tr_meulage_bavure_P283 :=[[136.49109375,-133.125578125,16],[0.60869059863804,-0.613253389411855,-0.357287378454986,0.354629052252209],[0,0,0,0],[8.999999E+09,8.999999E+09,8.999999E+09,8.999999E+09,8.999999E+09,8.999999E+09]];
	LOCAL CONST Robtarget Tr_meulage_bavure_P284 :=[[135.589421875,-134.34003125,16],[0.606809153742224,-0.610619816583659,-0.360934203724167,0.358681740700563],[0,0,0,0],[8.999999E+09,8.999999E+09,8.999999E+09,8.999999E+09,8.999999E+09,8.999999E+09]];
	LOCAL CONST Robtarget Tr_meulage_bavure_P285 :=[[134.770875,-135.49840625,16],[0.604187975688785,-0.607362877961505,-0.365692280383206,0.363780676473527],[0,0,0,0],[8.999999E+09,8.999999E+09,8.999999E+09,8.999999E+09,8.999999E+09,8.999999E+09]];
	LOCAL CONST Robtarget Tr_meulage_bavure_P286 :=[[133.573671875,-137.730640625,16],[0.601416707057644,-0.604070711573766,-0.370540372403093,0.368912391104014],[0,0,0,0],[8.999999E+09,8.999999E+09,8.999999E+09,8.999999E+09,8.999999E+09,8.999999E+09]];
	LOCAL CONST Robtarget Tr_meulage_bavure_P287 :=[[133.108828125,-139.018546875,16],[0.599140362240513,-0.601376565025791,-0.374444816355674,0.373052453250817],[0,0,0,0],[8.999999E+09,8.999999E+09,8.999999E+09,8.999999E+09,8.999999E+09,8.999999E+09]];
	LOCAL CONST Robtarget Tr_meulage_bavure_P288 :=[[132.29278125,-140.600125,16],[0.597729431643992,-0.599676521954628,-0.376847655033012,0.375624067997606],[0,0,0,0],[8.999999E+09,8.999999E+09,8.999999E+09,8.999999E+09,8.999999E+09,8.999999E+09]];
	LOCAL CONST Robtarget Tr_meulage_bavure_P289 :=[[131.3254375,-143.260328125,16],[0.597163392446936,-0.598937749449976,-0.377831999251129,0.376712669480281],[0,0,0,0],[8.999999E+09,8.999999E+09,8.999999E+09,8.999999E+09,8.999999E+09,8.999999E+09]];
	LOCAL CONST Robtarget Tr_meulage_bavure_P290 :=[[130.809875,-144.2653125,16],[0.597056893879946,-0.598761785707264,-0.378034432378165,0.376958031329215],[0,0,0,0],[8.999999E+09,8.999999E+09,8.999999E+09,8.999999E+09,8.999999E+09,8.999999E+09]];
	LOCAL CONST Robtarget Tr_meulage_bavure_P291 :=[[130.5497421875,-144.7399375,16],[0.596833034476496,-0.598559817524481,-0.378379007981161,0.377287423752542],[0,0,0,0],[8.999999E+09,8.999999E+09,8.999999E+09,8.999999E+09,8.999999E+09,8.999999E+09]];
	LOCAL CONST Robtarget Tr_meulage_bavure_P292 :=[[130.4254140625,-144.931609375,16],[0.595828133701051,-0.597663354216964,-0.379916045837112,0.378749453111081],[0,0,0,0],[8.999999E+09,8.999999E+09,8.999999E+09,8.999999E+09,8.999999E+09,8.999999E+09]];
	LOCAL CONST Robtarget Tr_meulage_bavure_P293 :=[[126.363828125,-152.60990625,16],[0.593014540964361,-0.595023303575851,-0.384237019461418,0.382939858570397],[0,0,0,0],[8.999999E+09,8.999999E+09,8.999999E+09,8.999999E+09,8.999999E+09,8.999999E+09]];
	LOCAL CONST Robtarget Tr_meulage_bavure_P294 :=[[126.017578125,-153.26628125,16],[0.58537258395462,-0.58758872306254,-0.395763616013899,0.394270961045354],[0,0,0,0],[8.999999E+09,8.999999E+09,8.999999E+09,8.999999E+09,8.999999E+09,8.999999E+09]];
	LOCAL CONST Robtarget Tr_meulage_bavure_P295 :=[[124.9164453125,-155.774171875,16],[0.551261408535918,-0.553617475186278,-0.442312222547626,0.440429845051792],[0,0,0,0],[8.999999E+09,8.999999E+09,8.999999E+09,8.999999E+09,8.999999E+09,8.999999E+09]];
	LOCAL CONST Robtarget Tr_meulage_bavure_P296 :=[[123.527890625,-158.6770625,16],[0.175884491247366,-0.176735690959794,0.686424365405069,-0.683118387878608],[0,0,0,0],[8.999999E+09,8.999999E+09,8.999999E+09,8.999999E+09,8.999999E+09,8.999999E+09]];
	LOCAL CONST Robtarget Tr_meulage_bavure_P297 :=[[123.327640625,-159.0216875,16],[0.306890262185601,-0.308559664737703,0.638359933428414,-0.63490621013334],[0,0,0,0],[8.999999E+09,8.999999E+09,8.999999E+09,8.999999E+09,8.999999E+09,8.999999E+09]];
	LOCAL CONST Robtarget Tr_meulage_bavure_P298 :=[[123.24621875,-159.1608125,16],[0.323837374309504,-0.325798370301669,0.629979367059983,-0.626187491082189],[0,0,0,0],[8.999999E+09,8.999999E+09,8.999999E+09,8.999999E+09,8.999999E+09,8.999999E+09]];
	LOCAL CONST Robtarget Tr_meulage_bavure_P299 :=[[123.3297109375,-159.02396875,16],[0.326372290266443,-0.328545755661438,0.628789577602118,-0.624629875752065],[0,0,0,0],[8.999999E+09,8.999999E+09,8.999999E+09,8.999999E+09,8.999999E+09,8.999999E+09]];
	LOCAL CONST Robtarget Tr_meulage_bavure_P300 :=[[123.180421875,-159.3618125,16],[0.317367343408428,-0.319672774505755,0.633583651159483,-0.629014342889801],[0,0,0,0],[8.999999E+09,8.999999E+09,8.999999E+09,8.999999E+09,8.999999E+09,8.999999E+09]];
	LOCAL CONST Robtarget Tr_meulage_bavure_P301 :=[[123.049625,-159.624921875,16],[0.226437807215411,-0.228206180781724,0.67216921894498,-0.666960568264265],[0,0,0,0],[8.999999E+09,8.999999E+09,8.999999E+09,8.999999E+09,8.999999E+09,8.999999E+09]];
	LOCAL CONST Robtarget Tr_meulage_bavure_P302 :=[[118.229125,-168.77559375,16],[0.57259715584048,-0.577338335268194,-0.413283646593551,0.409889706154571],[0,0,0,0],[8.999999E+09,8.999999E+09,8.999999E+09,8.999999E+09,8.999999E+09,8.999999E+09]];
	LOCAL CONST Robtarget Tr_meulage_bavure_P303 :=[[117.39971875,-170.24215625,16],[0.593299137055303,-0.598439080531331,-0.382339596409506,0.379055713424378],[0,0,0,0],[8.999999E+09,8.999999E+09,8.999999E+09,8.999999E+09,8.999999E+09,8.999999E+09]];
	LOCAL CONST Robtarget Tr_meulage_bavure_P304 :=[[116.6903671875,-171.53740625,16],[0.597199484310472,-0.602524035413321,-0.376035700168894,0.37271264385186],[0,0,0,0],[8.999999E+09,8.999999E+09,8.999999E+09,8.999999E+09,8.999999E+09,8.999999E+09]];
	LOCAL CONST Robtarget Tr_meulage_bavure_P305 :=[[115.400515625,-173.77928125,16],[0.597971590621077,-0.603355842809714,-0.374757996402828,0.371413715268589],[0,0,0,0],[8.999999E+09,8.999999E+09,8.999999E+09,8.999999E+09,8.999999E+09,8.999999E+09]];
	LOCAL CONST Robtarget Tr_meulage_bavure_P306 :=[[112.6163359375,-179.241234375,16],[0.597482480633576,-0.602809171466065,-0.375578015649989,0.372259240708357],[0,0,0,0],[8.999999E+09,8.999999E+09,8.999999E+09,8.999999E+09,8.999999E+09,8.999999E+09]];
	LOCAL CONST Robtarget Tr_meulage_bavure_P307 :=[[112.2888828125,-179.86715625,16],[0.59634366585415,-0.60148100378575,-0.377504189288559,0.374279870351197],[0,0,0,0],[8.999999E+09,8.999999E+09,8.999999E+09,8.999999E+09,8.999999E+09,8.999999E+09]];
	LOCAL CONST Robtarget Tr_meulage_bavure_P308 :=[[109.8376796875,-184.50940625,16],[0.59498469823415,-0.599775276329696,-0.379841033558747,0.376807133684962],[0,0,0,0],[8.999999E+09,8.999999E+09,8.999999E+09,8.999999E+09,8.999999E+09,8.999999E+09]];
	LOCAL CONST Robtarget Tr_meulage_bavure_P309 :=[[109.1857265625,-185.7065,16],[0.593876401343977,-0.598171387812109,-0.381829773780871,0.379088162020541],[0,0,0,0],[8.999999E+09,8.999999E+09,8.999999E+09,8.999999E+09,8.999999E+09,8.999999E+09]];
	LOCAL CONST Robtarget Tr_meulage_bavure_P310 :=[[108.3050546875,-187.32871875,16],[0.593535245767978,-0.597163793139388,-0.382678435768872,0.380353166139069],[0,0,0,0],[8.999999E+09,8.999999E+09,8.999999E+09,8.999999E+09,8.999999E+09,8.999999E+09]];
	LOCAL CONST Robtarget Tr_meulage_bavure_P311 :=[[105.85296875,-192.45959375,16],[0.59434502268286,-0.597119844745387,-0.3818072743853,0.38003301205267],[0,0,0,0],[8.999999E+09,8.999999E+09,8.999999E+09,8.999999E+09,8.999999E+09,8.999999E+09]];
	LOCAL CONST Robtarget Tr_meulage_bavure_P312 :=[[105.8435703125,-192.47709375,16],[0.596379963541565,-0.598112837284067,-0.379093326383236,0.377995003741926],[0,0,0,0],[8.999999E+09,8.999999E+09,8.999999E+09,8.999999E+09,8.999999E+09,8.999999E+09]];
	LOCAL CONST Robtarget Tr_meulage_bavure_P313 :=[[105.75275,-192.635765625,16],[0.599343028790232,-0.599854223923701,-0.374968253417973,0.374648705870072],[0,0,0,0],[8.999999E+09,8.999999E+09,8.999999E+09,8.999999E+09,8.999999E+09,8.999999E+09]];
	LOCAL CONST Robtarget Tr_meulage_bavure_P314 :=[[102.4508359375,-198.361921875,16],[0.602686810489317,-0.60178802922721,-0.370276878187595,0.370829893375242],[0,0,0,0],[8.999999E+09,8.999999E+09,8.999999E+09,8.999999E+09,8.999999E+09,8.999999E+09]];
	LOCAL CONST Robtarget Tr_meulage_bavure_P315 :=[[102.323703125,-198.554359375,16],[0.605820618133894,-0.603353526965027,-0.365956580905984,0.367452964383649],[0,0,0,0],[8.999999E+09,8.999999E+09,8.999999E+09,8.999999E+09,8.999999E+09,8.999999E+09]];
	LOCAL CONST Robtarget Tr_meulage_bavure_P316 :=[[102.198484375,-198.789375,16],[0.608366667680899,-0.604184152323163,-0.362646106408747,0.365156554429679],[0,0,0,0],[8.999999E+09,8.999999E+09,8.999999E+09,8.999999E+09,8.999999E+09,8.999999E+09]];
	LOCAL CONST Robtarget Tr_meulage_bavure_P317 :=[[99.5544765625,-203.31803125,16],[0.610259025865888,-0.604278225315239,-0.360449165247067,0.3640166851008],[0,0,0,0],[8.999999E+09,8.999999E+09,8.999999E+09,8.999999E+09,8.999999E+09,8.999999E+09]];
	LOCAL CONST Robtarget Tr_meulage_bavure_P318 :=[[98.0845625,-206.103328125,16],[0.611757304983226,-0.603942328844072,-0.358922765499279,0.363567203741494],[0,0,0,0],[8.999999E+09,8.999999E+09,8.999999E+09,8.999999E+09,8.999999E+09,8.999999E+09]];
	LOCAL CONST Robtarget Tr_meulage_bavure_P319 :=[[96.3557421875,-209.32040625,16],[0.613422733058156,-0.603759285474717,-0.357121868258397,0.362837769508845],[0,0,0,0],[8.999999E+09,8.999999E+09,8.999999E+09,8.999999E+09,8.999999E+09,8.999999E+09]];
	LOCAL CONST Robtarget Tr_meulage_bavure_P320 :=[[94.064328125,-213.881359375,16],[0.615973483698657,-0.604515851124367,-0.353798920659574,0.360504614200211],[0,0,0,0],[8.999999E+09,8.999999E+09,8.999999E+09,8.999999E+09,8.999999E+09,8.999999E+09]];
	LOCAL CONST Robtarget Tr_meulage_bavure_P321 :=[[93.3062734375,-215.341796875,16],[0.620223744935473,-0.607064343287252,-0.347493560353809,0.355026217116524],[0,0,0,0],[8.999999E+09,8.999999E+09,8.999999E+09,8.999999E+09,8.999999E+09,8.999999E+09]];
	LOCAL CONST Robtarget Tr_meulage_bavure_P322 :=[[92.51415625,-217.06746875,16],[0.626978657325296,-0.612225514490847,-0.336565402190736,0.344675808134505],[0,0,0,0],[8.999999E+09,8.999999E+09,8.999999E+09,8.999999E+09,8.999999E+09,8.999999E+09]];
	LOCAL CONST Robtarget Tr_meulage_bavure_P323 :=[[91.5088203125,-219.152453125,16],[0.636780633990478,-0.620601520657832,-0.319356513417838,0.327682154029593],[0,0,0,0],[8.999999E+09,8.999999E+09,8.999999E+09,8.999999E+09,8.999999E+09,8.999999E+09]];
	LOCAL CONST Robtarget Tr_meulage_bavure_P324 :=[[91.47390625,-219.191828125,16],[0.649759509928052,-0.632375845168603,-0.294185167913566,0.30227215664864],[0,0,0,0],[8.999999E+09,8.999999E+09,8.999999E+09,8.999999E+09,8.999999E+09,8.999999E+09]];
	LOCAL CONST Robtarget Tr_meulage_bavure_P325 :=[[89.031984375,-224.58059375,16],[0.665379634707229,-0.647106997433701,-0.259486185912631,0.266813408414437],[0,0,0,0],[8.999999E+09,8.999999E+09,8.999999E+09,8.999999E+09,8.999999E+09,8.999999E+09]];
	LOCAL CONST Robtarget Tr_meulage_bavure_P326 :=[[87.75640625,-225.97453125,16],[0.682283427897183,-0.663543222347988,-0.213982268941456,0.220025690935364],[0,0,0,0],[8.999999E+09,8.999999E+09,8.999999E+09,8.999999E+09,8.999999E+09,8.999999E+09]];
	LOCAL CONST Robtarget Tr_meulage_bavure_P327 :=[[86.6574375,-227.218390625,16],[0.698159810904856,-0.679509025705037,-0.157264217258917,0.161580717886219],[0,0,0,0],[8.999999E+09,8.999999E+09,8.999999E+09,8.999999E+09,8.999999E+09,8.999999E+09]];
	LOCAL CONST Robtarget Tr_meulage_bavure_P328 :=[[84.553984375,-227.948859375,16],[0.709928729567786,-0.692086094809517,-0.0910630247861073,0.0934107157792184],[0,0,0,0],[8.999999E+09,8.999999E+09,8.999999E+09,8.999999E+09,8.999999E+09,8.999999E+09]];
	LOCAL CONST Robtarget Tr_meulage_bavure_P329 :=[[83.169921875,-228.411015625,16],[0.714862807594626,-0.698661654609821,-0.020294528193253,0.0207651347505815],[0,0,0,0],[8.999999E+09,8.999999E+09,8.999999E+09,8.999999E+09,8.999999E+09,8.999999E+09]];
	LOCAL CONST Robtarget Tr_meulage_bavure_P330 :=[[81.2208828125,-227.939171875,16],[0.712309690921315,-0.698537708814796,0.0477964727712821,-0.0487388015238381],[0,0,0,0],[8.999999E+09,8.999999E+09,8.999999E+09,8.999999E+09,8.999999E+09,8.999999E+09]];
	LOCAL CONST Robtarget Tr_meulage_bavure_P331 :=[[80.7574453125,-227.8065625,16],[0.704174219667157,-0.693500810705246,0.106866858125182,-0.108511605562585],[0,0,0,0],[8.999999E+09,8.999999E+09,8.999999E+09,8.999999E+09,8.999999E+09,8.999999E+09]];
	LOCAL CONST Robtarget Tr_meulage_bavure_P332 :=[[80.7188125,-227.772203125,16],[0.693430784957216,-0.686413215994504,0.154114433581922,-0.155690027758446],[0,0,0,0],[8.999999E+09,8.999999E+09,8.999999E+09,8.999999E+09,8.999999E+09,8.999999E+09]];
	LOCAL CONST Robtarget Tr_meulage_bavure_P333 :=[[80.2228671875,-227.449640625,16],[0.682452893277903,-0.679533884544434,0.189975026189948,-0.190791083745285],[0,0,0,0],[8.999999E+09,8.999999E+09,8.999999E+09,8.999999E+09,8.999999E+09,8.999999E+09]];
	LOCAL CONST Robtarget Tr_meulage_bavure_P334 :=[[77.0405859375,-225.380796875,16],[0.672492316008928,-0.674019559820812,0.216406686197642,-0.215916335780462],[0,0,0,0],[8.999999E+09,8.999999E+09,8.999999E+09,8.999999E+09,8.999999E+09,8.999999E+09]];
	LOCAL CONST Robtarget Tr_meulage_bavure_P335 :=[[75.4690234375,-223.864234375,16],[0.663931197282134,-0.670218263904971,0.235626377130268,-0.233416054298293],[0,0,0,0],[8.999999E+09,8.999999E+09,8.999999E+09,8.999999E+09,8.999999E+09,8.999999E+09]];
	LOCAL CONST Robtarget Tr_meulage_bavure_P336 :=[[73.2680078125,-221.63965625,16],[0.656738916579173,-0.6680403392527,0.249504070467687,-0.245283141291052],[0,0,0,0],[8.999999E+09,8.999999E+09,8.999999E+09,8.999999E+09,8.999999E+09,8.999999E+09]];
	LOCAL CONST Robtarget Tr_meulage_bavure_P337 :=[[71.3517421875,-219.678125,16],[0.650709287432056,-0.667217421856874,0.259508734875249,-0.25308803160912],[0,0,0,0],[8.999999E+09,8.999999E+09,8.999999E+09,8.999999E+09,8.999999E+09,8.999999E+09]];
	LOCAL CONST Robtarget Tr_meulage_bavure_P338 :=[[68.4788828125,-216.646171875,16],[0.645605859980727,-0.667426078138494,0.266750885905939,-0.258029976257819],[0,0,0,0],[8.999999E+09,8.999999E+09,8.999999E+09,8.999999E+09,8.999999E+09,8.999999E+09]];
	LOCAL CONST Robtarget Tr_meulage_bavure_P339 :=[[66.046109375,-214.186734375,16],[0.641160073186351,-0.668333390187963,0.272162748699046,-0.261097066877658],[0,0,0,0],[8.999999E+09,8.999999E+09,8.999999E+09,8.999999E+09,8.999999E+09,8.999999E+09]];
	LOCAL CONST Robtarget Tr_meulage_bavure_P340 :=[[65.36596875,-213.47665625,16],[0.637108723768627,-0.669593983653222,0.276566491563365,-0.263148906320455],[0,0,0,0],[8.999999E+09,8.999999E+09,8.999999E+09,8.999999E+09,8.999999E+09,8.999999E+09]];
	LOCAL CONST Robtarget Tr_meulage_bavure_P341 :=[[59.7366328125,-208.055453125,16],[0.633276837453571,-0.670929708244459,0.280534510113967,-0.264790789822694],[0,0,0,0],[8.999999E+09,8.999999E+09,8.999999E+09,8.999999E+09,8.999999E+09,8.999999E+09]];
	LOCAL CONST Robtarget Tr_meulage_bavure_P342 :=[[59.5100703125,-207.82415625,16],[0.629576317677475,-0.672176177841971,0.284375077770646,-0.26635251323081],[0,0,0,0],[8.999999E+09,8.999999E+09,8.999999E+09,8.999999E+09,8.999999E+09,8.999999E+09]];
	LOCAL CONST Robtarget Tr_meulage_bavure_P343 :=[[56.99353125,-205.091140625,16],[0.626045160067526,-0.673303743302813,0.288071157986889,-0.267851702900202],[0,0,0,0],[8.999999E+09,8.999999E+09,8.999999E+09,8.999999E+09,8.999999E+09,8.999999E+09]];
	LOCAL CONST Robtarget Tr_meulage_bavure_P344 :=[[52.645171875,-200.83184375,16],[0.622822930646747,-0.674414105025693,0.291329463033691,-0.26904340908391],[0,0,0,0],[8.999999E+09,8.999999E+09,8.999999E+09,8.999999E+09,8.999999E+09,8.999999E+09]];
	LOCAL CONST Robtarget Tr_meulage_bavure_P345 :=[[51.76696875,-199.84040625,16],[0.620105972019481,-0.675653889369191,0.293738275373029,-0.269589003534898],[0,0,0,0],[8.999999E+09,8.999999E+09,8.999999E+09,8.999999E+09,8.999999E+09,8.999999E+09]];
	LOCAL CONST Robtarget Tr_meulage_bavure_P346 :=[[50.91873046875,-198.992203125,16],[0.618031319622084,-0.677139937837452,0.294998870041727,-0.269247951200713],[0,0,0,0],[8.999999E+09,8.999999E+09,8.999999E+09,8.999999E+09,8.999999E+09,8.999999E+09]];
	LOCAL CONST Robtarget Tr_meulage_bavure_P347 :=[[49.6188984375,-197.668390625,16],[0.616620799214955,-0.678884639262754,0.295070012513416,-0.268007694411788],[0,0,0,0],[8.999999E+09,8.999999E+09,8.999999E+09,8.999999E+09,8.999999E+09,8.999999E+09]];
	LOCAL CONST Robtarget Tr_meulage_bavure_P348 :=[[45.7632734375,-193.478296875,16],[0.61580087689486,-0.6807781059835,0.294159800919224,-0.266083561972931],[0,0,0,0],[8.999999E+09,8.999999E+09,8.999999E+09,8.999999E+09,8.999999E+09,8.999999E+09]];
	LOCAL CONST Robtarget Tr_meulage_bavure_P349 :=[[42.14279296875,-189.82240625,16],[0.615431201670511,-0.682644945442827,0.292637882671618,-0.263824532781209],[0,0,0,0],[8.999999E+09,8.999999E+09,8.999999E+09,8.999999E+09,8.999999E+09,8.999999E+09]];
	LOCAL CONST Robtarget Tr_meulage_bavure_P350 :=[[41.9723515625,-189.659125,16],[0.615363957239353,-0.6843320735089,0.29087009788068,-0.261555729160377],[0,0,0,0],[8.999999E+09,8.999999E+09,8.999999E+09,8.999999E+09,8.999999E+09,8.999999E+09]];
	LOCAL CONST Robtarget Tr_meulage_bavure_P351 :=[[41.7776171875,-189.454765625,16],[0.615527994340268,-0.685735953657101,0.289073111632725,-0.259476831675601],[0,0,0,0],[8.999999E+09,8.999999E+09,8.999999E+09,8.999999E+09,8.999999E+09,8.999999E+09]];
	LOCAL CONST Robtarget Tr_meulage_bavure_P352 :=[[38.5902109375,-186.12478125,16],[0.615889930140434,-0.686855731074871,0.287301342831601,-0.257617423805873],[0,0,0,0],[8.999999E+09,8.999999E+09,8.999999E+09,8.999999E+09,8.999999E+09,8.999999E+09]];
	LOCAL CONST Robtarget Tr_meulage_bavure_P353 :=[[34.9079296875,-182.3803125,16],[0.616467040633372,-0.687728842297101,0.285493966701297,-0.255911356259506],[0,0,0,0],[8.999999E+09,8.999999E+09,8.999999E+09,8.999999E+09,8.999999E+09,8.999999E+09]];
	LOCAL CONST Robtarget Tr_meulage_bavure_P354 :=[[34.7763984375,-182.24615625,16],[0.617291071587836,-0.688375449548463,0.283586543321303,-0.254302272589071],[0,0,0,0],[8.999999E+09,8.999999E+09,8.999999E+09,8.999999E+09,8.999999E+09,8.999999E+09]];
	LOCAL CONST Robtarget Tr_meulage_bavure_P355 :=[[32.5143125,-180.000421875,16],[0.6183132434262,-0.688812829130285,0.281629630911457,-0.252805004740772],[0,0,0,0],[8.999999E+09,8.999999E+09,8.999999E+09,8.999999E+09,8.999999E+09,8.999999E+09]];
	LOCAL CONST Robtarget Tr_meulage_bavure_P356 :=[[31.0621328125,-178.407890625,16],[0.619464540090699,-0.688979568537382,0.279795685122259,-0.251565522866761],[0,0,0,0],[8.999999E+09,8.999999E+09,8.999999E+09,8.999999E+09,8.999999E+09,8.999999E+09]];
	LOCAL CONST Robtarget Tr_meulage_bavure_P357 :=[[28.63885546875,-175.808015625,16],[0.620623324488447,-0.68878816209319,0.278366282189568,-0.250818200697539],[0,0,0,0],[8.999999E+09,8.999999E+09,8.999999E+09,8.999999E+09,8.999999E+09,8.999999E+09]];
	LOCAL CONST Robtarget Tr_meulage_bavure_P358 :=[[26.3606875,-173.6865,16],[0.621659771460173,-0.68814685167237,0.277640849716816,-0.250815864031794],[0,0,0,0],[8.999999E+09,8.999999E+09,8.999999E+09,8.999999E+09,8.999999E+09,8.999999E+09]];
	LOCAL CONST Robtarget Tr_meulage_bavure_P359 :=[[26.3401796875,-173.665375,16],[0.622466331881606,-0.686988207236225,0.27785196952162,-0.251756135625675],[0,0,0,0],[8.999999E+09,8.999999E+09,8.999999E+09,8.999999E+09,8.999999E+09,8.999999E+09]];
	LOCAL CONST Robtarget Tr_meulage_bavure_P360 :=[[23.891693359375,-170.99246875,16],[0.622957887826191,-0.685297436536254,0.279124301910439,-0.253733162111264],[0,0,0,0],[8.999999E+09,8.999999E+09,8.999999E+09,8.999999E+09,8.999999E+09,8.999999E+09]];
	LOCAL CONST Robtarget Tr_meulage_bavure_P361 :=[[22.627533203125,-169.7788125,16],[0.623115669025229,-0.683101151946932,0.28142359324525,-0.256710810814327],[0,0,0,0],[8.999999E+09,8.999999E+09,8.999999E+09,8.999999E+09,8.999999E+09,8.999999E+09]];
	LOCAL CONST Robtarget Tr_meulage_bavure_P362 :=[[20.934509765625,-167.98546875,16],[0.622968611368631,-0.680492557087961,0.284562448019971,-0.260507585636598],[0,0,0,0],[8.999999E+09,8.999999E+09,8.999999E+09,8.999999E+09,8.999999E+09,8.999999E+09]];
	LOCAL CONST Robtarget Tr_meulage_bavure_P363 :=[[18.89404296875,-165.9073125,16],[0.62259227075011,-0.677641481659719,0.288208607502964,-0.264795553772049],[0,0,0,0],[8.999999E+09,8.999999E+09,8.999999E+09,8.999999E+09,8.999999E+09,8.999999E+09]];
	LOCAL CONST Robtarget Tr_meulage_bavure_P364 :=[[13.930755859375,-160.69478125,16],[0.622132867085854,-0.674766908434734,0.291903052276922,-0.269133652753392],[0,0,0,0],[8.999999E+09,8.999999E+09,8.999999E+09,8.999999E+09,8.999999E+09,8.999999E+09]];
	LOCAL CONST Robtarget Tr_meulage_bavure_P365 :=[[11.089203125,-157.940328125,16],[0.62176380044021,-0.672131047995704,0.29514031462928,-0.273023488848254],[0,0,0,0],[8.999999E+09,8.999999E+09,8.999999E+09,8.999999E+09,8.999999E+09,8.999999E+09]];
	LOCAL CONST Robtarget Tr_meulage_bavure_P366 :=[[9.912048828125,-156.8128125,16],[0.621683349370595,-0.669970923925728,0.297440874260378,-0.27600308065072],[0,0,0,0],[8.999999E+09,8.999999E+09,8.999999E+09,8.999999E+09,8.999999E+09,8.999999E+09]];
	LOCAL CONST Robtarget Tr_meulage_bavure_P367 :=[[8.3047177734375,-155.029109375,16],[0.622023253974866,-0.668486346339496,0.298467876118716,-0.277722889221204],[0,0,0,0],[8.999999E+09,8.999999E+09,8.999999E+09,8.999999E+09,8.999999E+09,8.999999E+09]];
	LOCAL CONST Robtarget Tr_meulage_bavure_P368 :=[[7.17446875,-153.708140625,16],[0.622828898193416,-0.667780453097403,0.298088543319346,-0.278022751547339],[0,0,0,0],[8.999999E+09,8.999999E+09,8.999999E+09,8.999999E+09,8.999999E+09,8.999999E+09]];
	LOCAL CONST Robtarget Tr_meulage_bavure_P369 :=[[6.1098935546875,-152.56575,16],[0.624058575301547,-0.667829769104241,0.296388445215739,-0.276962422782181],[0,0,0,0],[8.999999E+09,8.999999E+09,8.999999E+09,8.999999E+09,8.999999E+09,8.999999E+09]];
	LOCAL CONST Robtarget Tr_meulage_bavure_P370 :=[[2.68130493164063,-148.779546875,16],[0.625564563355642,-0.668504788856882,0.293678690378308,-0.274814757912966],[0,0,0,0],[8.999999E+09,8.999999E+09,8.999999E+09,8.999999E+09,8.999999E+09,8.999999E+09]];
	LOCAL CONST Robtarget Tr_meulage_bavure_P371 :=[[1.38775634765625,-147.379734375,16],[0.627144830944035,-0.669598032763958,0.290416524721506,-0.27200381928844],[0,0,0,0],[8.999999E+09,8.999999E+09,8.999999E+09,8.999999E+09,8.999999E+09,8.999999E+09]];
	LOCAL CONST Robtarget Tr_meulage_bavure_P372 :=[[-1.8812255859375,-144.168984375,16],[0.628573054108754,-0.670884385790244,0.287124405095647,-0.269016045152909],[0,0,0,0],[8.999999E+09,8.999999E+09,8.999999E+09,8.999999E+09,8.999999E+09,8.999999E+09]];
	LOCAL CONST Robtarget Tr_meulage_bavure_P373 :=[[-2.87652587890625,-143.143890625,16],[0.629658597769557,-0.67216514592231,0.284272372338623,-0.266295484729063],[0,0,0,0],[8.999999E+09,8.999999E+09,8.999999E+09,8.999999E+09,8.999999E+09,8.999999E+09]];
	LOCAL CONST Robtarget Tr_meulage_bavure_P374 :=[[-3.07424926757813,-142.944234375,16],[0.630296551734283,-0.673297000267911,0.282172611197929,-0.264151516732058],[0,0,0,0],[8.999999E+09,8.999999E+09,8.999999E+09,8.999999E+09,8.999999E+09,8.999999E+09]];
	LOCAL CONST Robtarget Tr_meulage_bavure_P375 :=[[-5.2728271484375,-140.780734375,16],[0.630445176015824,-0.674236008882384,0.280949155416218,-0.262701839421888],[0,0,0,0],[8.999999E+09,8.999999E+09,8.999999E+09,8.999999E+09,8.999999E+09,8.999999E+09]];
	LOCAL CONST Robtarget Tr_meulage_bavure_P376 :=[[-7.9797666015625,-137.97146875,16],[0.630172281736214,-0.675001580719101,0.280499144265552,-0.261870180479529],[0,0,0,0],[8.999999E+09,8.999999E+09,8.999999E+09,8.999999E+09,8.999999E+09,8.999999E+09]];
	LOCAL CONST Robtarget Tr_meulage_bavure_P377 :=[[-9.6129453125,-136.363828125,16],[0.629602643090359,-0.675682367399799,0.280556270063144,-0.26142308529832],[0,0,0,0],[8.999999E+09,8.999999E+09,8.999999E+09,8.999999E+09,8.999999E+09,8.999999E+09]];
	LOCAL CONST Robtarget Tr_meulage_bavure_P378 :=[[-10.7795107421875,-135.26734375,16],[0.628898604778399,-0.676425966058553,0.280731339055059,-0.261006460881508],[0,0,0,0],[8.999999E+09,8.999999E+09,8.999999E+09,8.999999E+09,8.999999E+09,8.999999E+09]];
	LOCAL CONST Robtarget Tr_meulage_bavure_P379 :=[[-13.36590625,-132.63265625,16],[0.628262031678337,-0.677401563078235,0.280552249035713,-0.260200648445724],[0,0,0,0],[8.999999E+09,8.999999E+09,8.999999E+09,8.999999E+09,8.999999E+09,8.999999E+09]];
	LOCAL CONST Robtarget Tr_meulage_bavure_P380 :=[[-14.297515625,-131.754234375,16],[0.627888226714868,-0.678754928570377,0.279574923893112,-0.258623246488867],[0,0,0,0],[8.999999E+09,8.999999E+09,8.999999E+09,8.999999E+09,8.999999E+09,8.999999E+09]];
	LOCAL CONST Robtarget Tr_meulage_bavure_P381 :=[[-15.38885546875,-130.5290546875,16],[0.627902487479892,-0.680570709147324,0.277506869054569,-0.256031079548563],[0,0,0,0],[8.999999E+09,8.999999E+09,8.999999E+09,8.999999E+09,8.999999E+09,8.999999E+09]];
	LOCAL CONST Robtarget Tr_meulage_bavure_P382 :=[[-16.74499609375,-129.1134921875,16],[0.628302395955882,-0.682810958563061,0.274356916082425,-0.252455098383917],[0,0,0,0],[8.999999E+09,8.999999E+09,8.999999E+09,8.999999E+09,8.999999E+09,8.999999E+09]];
	LOCAL CONST Robtarget Tr_meulage_bavure_P383 :=[[-17.981017578125,-127.745984375,16],[0.628939494300714,-0.685288143347013,0.270513126360756,-0.248269856332369],[0,0,0,0],[8.999999E+09,8.999999E+09,8.999999E+09,8.999999E+09,8.999999E+09,8.999999E+09]];
	LOCAL CONST Robtarget Tr_meulage_bavure_P384 :=[[-20.975953125,-124.5475625,16],[0.629585224954973,-0.68768788695737,0.266660852834262,-0.244130711333514],[0,0,0,0],[8.999999E+09,8.999999E+09,8.999999E+09,8.999999E+09,8.999999E+09,8.999999E+09]];
	LOCAL CONST Robtarget Tr_meulage_bavure_P385 :=[[-21.87841796875,-123.8248125,16],[0.6299753179832,-0.689705613850408,0.263580726862804,-0.240753951954425],[0,0,0,0],[8.999999E+09,8.999999E+09,8.999999E+09,8.999999E+09,8.999999E+09,8.999999E+09]];
	LOCAL CONST Robtarget Tr_meulage_bavure_P386 :=[[-23.670623046875,-121.965,16],[0.629955032695945,-0.69113538767018,0.261807688703997,-0.238632074178036],[0,0,0,0],[8.999999E+09,8.999999E+09,8.999999E+09,8.999999E+09,8.999999E+09,8.999999E+09]];
	LOCAL CONST Robtarget Tr_meulage_bavure_P387 :=[[-24.449462890625,-121.1865078125,16],[0.629520296521883,-0.691950467182103,0.261423582490461,-0.237837040326613],[0,0,0,0],[8.999999E+09,8.999999E+09,8.999999E+09,8.999999E+09,8.999999E+09,8.999999E+09]];
	LOCAL CONST Robtarget Tr_meulage_bavure_P388 :=[[-26.42593359375,-119.3252734375,16],[0.628820332090553,-0.69230429897565,0.262024861767564,-0.23799730961725],[0,0,0,0],[8.999999E+09,8.999999E+09,8.999999E+09,8.999999E+09,8.999999E+09,8.999999E+09]];
	LOCAL CONST Robtarget Tr_meulage_bavure_P389 :=[[-28.22183203125,-117.755125,16],[0.62811302891453,-0.692465557667882,0.262881271165393,-0.238451067563119],[0,0,0,0],[8.999999E+09,8.999999E+09,8.999999E+09,8.999999E+09,8.999999E+09,8.999999E+09]];
	LOCAL CONST Robtarget Tr_meulage_bavure_P390 :=[[-29.665802734375,-116.402390625,16],[0.627657667039363,-0.692715252727711,0.263245850746348,-0.238522648211693],[0,0,0,0],[8.999999E+09,8.999999E+09,8.999999E+09,8.999999E+09,8.999999E+09,8.999999E+09]];
	LOCAL CONST Robtarget Tr_meulage_bavure_P391 :=[[-30.951232421875,-115.1545234375,16],[0.627629146482942,-0.693245668825777,0.262611345104371,-0.237754870742677],[0,0,0,0],[8.999999E+09,8.999999E+09,8.999999E+09,8.999999E+09,8.999999E+09,8.999999E+09]];
	LOCAL CONST Robtarget Tr_meulage_bavure_P392 :=[[-32.138244140625,-114.108234375,16],[0.628047909231153,-0.694098819930288,0.260882695846487,-0.236056922986022],[0,0,0,0],[8.999999E+09,8.999999E+09,8.999999E+09,8.999999E+09,8.999999E+09,8.999999E+09]];
	LOCAL CONST Robtarget Tr_meulage_bavure_P393 :=[[-33.7190859375,-112.4650703125,16],[0.628802945731713,-0.695155391901145,0.258360478193116,-0.233700021090519],[0,0,0,0],[8.999999E+09,8.999999E+09,8.999999E+09,8.999999E+09,8.999999E+09,8.999999E+09]];
	LOCAL CONST Robtarget Tr_meulage_bavure_P394 :=[[-37.08410546875,-109.042375,16],[0.629696429942186,-0.696186101434912,0.255629814310127,-0.231215735456507],[0,0,0,0],[8.999999E+09,8.999999E+09,8.999999E+09,8.999999E+09,8.999999E+09,8.999999E+09]];
	LOCAL CONST Robtarget Tr_meulage_bavure_P395 :=[[-38.87545703125,-107.05653125,16],[0.630481901785135,-0.696935375574078,0.253413026850777,-0.229249845402665],[0,0,0,0],[8.999999E+09,8.999999E+09,8.999999E+09,8.999999E+09,8.999999E+09,8.999999E+09]];
	LOCAL CONST Robtarget Tr_meulage_bavure_P396 :=[[-40.1063828125,-105.6612578125,16],[0.630948083935846,-0.697187971913402,0.252347981679493,-0.22837237866968],[0,0,0,0],[8.999999E+09,8.999999E+09,8.999999E+09,8.999999E+09,8.999999E+09,8.999999E+09]];
	LOCAL CONST Robtarget Tr_meulage_bavure_P397 :=[[-40.53662109375,-105.322171875,16],[0.630969976008754,-0.696803480866971,0.25283432956057,-0.228946719179032],[0,0,0,0],[8.999999E+09,8.999999E+09,8.999999E+09,8.999999E+09,8.999999E+09,8.999999E+09]];
	LOCAL CONST Robtarget Tr_meulage_bavure_P398 :=[[-42.30416796875,-103.549515625,16],[0.630508668929816,-0.695753325807529,0.254956736705307,-0.231048026264444],[0,0,0,0],[8.999999E+09,8.999999E+09,8.999999E+09,8.999999E+09,8.999999E+09,8.999999E+09]];
	LOCAL CONST Robtarget Tr_meulage_bavure_P399 :=[[-42.6742265625,-102.88034375,16],[0.629619958517586,-0.694114329208192,0.258479120006028,-0.234462257826468],[0,0,0,0],[8.999999E+09,8.999999E+09,8.999999E+09,8.999999E+09,8.999999E+09,8.999999E+09]];
	LOCAL CONST Robtarget Tr_meulage_bavure_P400 :=[[-43.97119140625,-101.8010390625,16],[0.628438935361893,-0.692048700393345,0.262922981827168,-0.238756374642025],[0,0,0,0],[8.999999E+09,8.999999E+09,8.999999E+09,8.999999E+09,8.999999E+09,8.999999E+09]];
	LOCAL CONST Robtarget Tr_meulage_bavure_P401 :=[[-44.6539609375,-100.9943828125,16],[0.627142620083092,-0.689777066550819,0.26769680558972,-0.243388892131342],[0,0,0,0],[8.999999E+09,8.999999E+09,8.999999E+09,8.999999E+09,8.999999E+09,8.999999E+09]];
	LOCAL CONST Robtarget Tr_meulage_bavure_P402 :=[[-45.29446484375,-100.1923671875,16],[0.625936858366737,-0.687552353768805,0.272173741068197,-0.247782696808911],[0,0,0,0],[8.999999E+09,8.999999E+09,8.999999E+09,8.999999E+09,8.999999E+09,8.999999E+09]];
	LOCAL CONST Robtarget Tr_meulage_bavure_P403 :=[[-47.58019921875,-98.0126171875,16],[0.62504449146584,-0.685642452462711,0.275734568137808,-0.251364792687808],[0,0,0,0],[8.999999E+09,8.999999E+09,8.999999E+09,8.999999E+09,8.999999E+09,8.999999E+09]];
	LOCAL CONST Robtarget Tr_meulage_bavure_P404 :=[[-51.10696484375,-94.6501484375,16],[0.624675603163293,-0.684309926059204,0.277818699792386,-0.253608134639035],[0,0,0,0],[8.999999E+09,8.999999E+09,8.999999E+09,8.999999E+09,8.999999E+09,8.999999E+09]];
	LOCAL CONST Robtarget Tr_meulage_bavure_P405 :=[[-54.89083984375,-90.9807265625,16],[0.624986982684058,-0.683766731129888,0.278002534250303,-0.254104151532071],[0,0,0,0],[8.999999E+09,8.999999E+09,8.999999E+09,8.999999E+09,8.999999E+09,8.999999E+09]];
	LOCAL CONST Robtarget Tr_meulage_bavure_P406 :=[[-54.9040546875,-90.9685078125,16],[0.626019696901709,-0.684095286415799,0.276143664093821,-0.252700722150962],[0,0,0,0],[8.999999E+09,8.999999E+09,8.999999E+09,8.999999E+09,8.999999E+09,8.999999E+09]];
	LOCAL CONST Robtarget Tr_meulage_bavure_P407 :=[[-54.91623046875,-90.9553046875,16],[0.627659701486804,-0.685198513711173,0.272481389711635,-0.249600056486995],[0,0,0,0],[8.999999E+09,8.999999E+09,8.999999E+09,8.999999E+09,8.999999E+09,8.999999E+09]];
	LOCAL CONST Robtarget Tr_meulage_bavure_P408 :=[[-58.02874609375,-87.6899375,16],[0.629643465233333,-0.686833771223962,0.267618136465409,-0.245334486833818],[0,0,0,0],[8.999999E+09,8.999999E+09,8.999999E+09,8.999999E+09,8.999999E+09,8.999999E+09]];
	LOCAL CONST Robtarget Tr_meulage_bavure_P409 :=[[-59.8401796875,-86.2268046875,16],[0.631653340102787,-0.688700026249457,0.262330690799729,-0.240601206242877],[0,0,0,0],[8.999999E+09,8.999999E+09,8.999999E+09,8.999999E+09,8.999999E+09,8.999999E+09]];
	LOCAL CONST Robtarget Tr_meulage_bavure_P410 :=[[-61.13094921875,-85.1266328125,16],[0.633442342231833,-0.690540011578096,0.257293874142449,-0.236019392860718],[0,0,0,0],[8.999999E+09,8.999999E+09,8.999999E+09,8.999999E+09,8.999999E+09,8.999999E+09]];
	LOCAL CONST Robtarget Tr_meulage_bavure_P411 :=[[-61.7408125,-84.5056484375,16],[0.634875965824457,-0.692246094761999,0.252870891932948,-0.231914131346625],[0,0,0,0],[8.999999E+09,8.999999E+09,8.999999E+09,8.999999E+09,8.999999E+09,8.999999E+09]];
	LOCAL CONST Robtarget Tr_meulage_bavure_P412 :=[[-64.62542578125,-81.7070625,16],[0.635948124143437,-0.693825099661232,0.249095126889814,-0.228316298669787],[0,0,0,0],[8.999999E+09,8.999999E+09,8.999999E+09,8.999999E+09,8.999999E+09,8.999999E+09]];
	LOCAL CONST Robtarget Tr_meulage_bavure_P413 :=[[-68.5583828125,-78.153609375,16],[0.636728417308657,-0.695348025745214,0.24578905059607,-0.225068408025045],[0,0,0,0],[8.999999E+09,8.999999E+09,8.999999E+09,8.999999E+09,8.999999E+09,8.999999E+09]];
	LOCAL CONST Robtarget Tr_meulage_bavure_P414 :=[[-69.5910625,-77.24471875,16],[0.637290882228162,-0.696895516977302,0.242739664872587,-0.221978433509507],[0,0,0,0],[8.999999E+09,8.999999E+09,8.999999E+09,8.999999E+09,8.999999E+09,8.999999E+09]];
	LOCAL CONST Robtarget Tr_meulage_bavure_P415 :=[[-70.2184453125,-76.72796875,16],[0.637695904333486,-0.698522585711101,0.239778170014126,-0.218898515372882],[0,0,0,0],[8.999999E+09,8.999999E+09,8.999999E+09,8.999999E+09,8.999999E+09,8.999999E+09]];
	LOCAL CONST Robtarget Tr_meulage_bavure_P416 :=[[-75.3584609375,-72.507171875,16],[0.638018287536529,-0.700268152875391,0.236724939723641,-0.215681435803552],[0,0,0,0],[8.999999E+09,8.999999E+09,8.999999E+09,8.999999E+09,8.999999E+09,8.999999E+09]];
	LOCAL CONST Robtarget Tr_meulage_bavure_P417 :=[[-78.0387890625,-70.51425,16],[0.638353066813411,-0.702185612103137,0.233333944908473,-0.212122602281571],[0,0,0,0],[8.999999E+09,8.999999E+09,8.999999E+09,8.999999E+09,8.999999E+09,8.999999E+09]];
	LOCAL CONST Robtarget Tr_meulage_bavure_P418 :=[[-78.582734375,-70.055484375,16],[0.638821305610421,-0.704357335734337,0.229252283366428,-0.207921796997581],[0,0,0,0],[8.999999E+09,8.999999E+09,8.999999E+09,8.999999E+09,8.999999E+09,8.999999E+09]];
	LOCAL CONST Robtarget Tr_meulage_bavure_P419 :=[[-79.387265625,-69.5151640625,16],[0.639517950907346,-0.706858831601742,0.224147613461056,-0.202793565069511],[0,0,0,0],[8.999999E+09,8.999999E+09,8.999999E+09,8.999999E+09,8.999999E+09,8.999999E+09]];
	LOCAL CONST Robtarget Tr_meulage_bavure_P420 :=[[-81.9696328125,-67.542171875,16],[0.640516788402793,-0.70969108392872,0.217799851836193,-0.196570683740947],[0,0,0,0],[8.999999E+09,8.999999E+09,8.999999E+09,8.999999E+09,8.999999E+09,8.999999E+09]];
	LOCAL CONST Robtarget Tr_meulage_bavure_P421 :=[[-88.5744921875,-63.05772265625,16],[0.641817352432653,-0.712779757314828,0.210209420404658,-0.189281544931598],[0,0,0,0],[8.999999E+09,8.999999E+09,8.999999E+09,8.999999E+09,8.999999E+09,8.999999E+09]];
	LOCAL CONST Robtarget Tr_meulage_bavure_P422 :=[[-91.1654375,-61.232359375,16],[0.643351213588247,-0.716000472563905,0.20158163914079,-0.181128081820868],[0,0,0,0],[8.999999E+09,8.999999E+09,8.999999E+09,8.999999E+09,8.999999E+09,8.999999E+09]];
	LOCAL CONST Robtarget Tr_meulage_bavure_P423 :=[[-92.53265625,-60.3967421875,16],[0.645049958046779,-0.719216920086579,0.192173865636861,-0.172356545716169],[0,0,0,0],[8.999999E+09,8.999999E+09,8.999999E+09,8.999999E+09,8.999999E+09,8.999999E+09]];
	LOCAL CONST Robtarget Tr_meulage_bavure_P424 :=[[-93.8419765625,-59.67143359375,16],[0.646866346859878,-0.722328260362969,0.182178670006239,-0.163146393695728],[0,0,0,0],[8.999999E+09,8.999999E+09,8.999999E+09,8.999999E+09,8.999999E+09,8.999999E+09]];
	LOCAL CONST Robtarget Tr_meulage_bavure_P425 :=[[-95.9725,-58.5518203125,16],[0.648791452895745,-0.725266269824136,0.171677483783545,-0.153575160968702],[0,0,0,0],[8.999999E+09,8.999999E+09,8.999999E+09,8.999999E+09,8.999999E+09,8.999999E+09]];
	LOCAL CONST Robtarget Tr_meulage_bavure_P426 :=[[-97.1642421875,-57.97534375,16],[0.650830083356341,-0.727988110881948,0.160680299605587,-0.143650110795537],[0,0,0,0],[8.999999E+09,8.999999E+09,8.999999E+09,8.999999E+09,8.999999E+09,8.999999E+09]];
	LOCAL CONST Robtarget Tr_meulage_bavure_P427 :=[[-98.99365625,-57.1351484375,16],[0.65297111138381,-0.730464859184432,0.149202207661245,-0.133373604674503],[0,0,0,0],[8.999999E+09,8.999999E+09,8.999999E+09,8.999999E+09,8.999999E+09,8.999999E+09]];
	LOCAL CONST Robtarget Tr_meulage_bavure_P428 :=[[-100.6922890625,-56.42620703125,16],[0.655201720288885,-0.732644994008814,0.137328546307158,-0.122812413271112],[0,0,0,0],[8.999999E+09,8.999999E+09,8.999999E+09,8.999999E+09,8.999999E+09,8.999999E+09]];
	LOCAL CONST Robtarget Tr_meulage_bavure_P429 :=[[-102.61703125,-55.6012109375,16],[0.657478845058019,-0.734485139373702,0.125239079520433,-0.112108524659106],[0,0,0,0],[8.999999E+09,8.999999E+09,8.999999E+09,8.999999E+09,8.999999E+09,8.999999E+09]];
	LOCAL CONST Robtarget Tr_meulage_bavure_P430 :=[[-104.8251953125,-54.848921875,16],[0.65976108123265,-0.735928135669543,0.1132290051315,-0.101510035058641],[0,0,0,0],[8.999999E+09,8.999999E+09,8.999999E+09,8.999999E+09,8.999999E+09,8.999999E+09]];
	LOCAL CONST Robtarget Tr_meulage_bavure_P431 :=[[-106.0003984375,-54.43116796875,16],[0.661999996344206,-0.736937670225042,0.101671806796521,-0.0913330101676741],[0,0,0,0],[8.999999E+09,8.999999E+09,8.999999E+09,8.999999E+09,8.999999E+09,8.999999E+09]];
	LOCAL CONST Robtarget Tr_meulage_bavure_P432 :=[[-108.479953125,-53.8170625,16],[0.664152456171227,-0.737505159043295,0.0909726979806991,-0.0819244991950728],[0,0,0,0],[8.999999E+09,8.999999E+09,8.999999E+09,8.999999E+09,8.999999E+09,8.999999E+09]];
	LOCAL CONST Robtarget Tr_meulage_bavure_P433 :=[[-110.90090625,-53.23883203125,16],[0.666210870070013,-0.737645385266296,0.0814393522814772,-0.0735526620583337],[0,0,0,0],[8.999999E+09,8.999999E+09,8.999999E+09,8.999999E+09,8.999999E+09,8.999999E+09]];
	LOCAL CONST Robtarget Tr_meulage_bavure_P434 :=[[-112.207796875,-53.0146796875,16],[0.668178460521285,-0.737424392634405,0.0731451634212463,-0.066276655854557],[0,0,0,0],[8.999999E+09,8.999999E+09,8.999999E+09,8.999999E+09,8.999999E+09,8.999999E+09]];
	LOCAL CONST Robtarget Tr_meulage_bavure_P435 :=[[-120.3569921875,-51.347,16],[0.670081415582182,-0.736931386684076,0.0658566991970994,-0.0598825766156174],[0,0,0,0],[8.999999E+09,8.999999E+09,8.999999E+09,8.999999E+09,8.999999E+09,8.999999E+09]];
	LOCAL CONST Robtarget Tr_meulage_bavure_P436 :=[[-121.9906015625,-51.03771875,16],[0.671955768223622,-0.736257924857006,0.059088695081722,-0.0539280979619761],[0,0,0,0],[8.999999E+09,8.999999E+09,8.999999E+09,8.999999E+09,8.999999E+09,8.999999E+09]];
	LOCAL CONST Robtarget Tr_meulage_bavure_P437 :=[[-122.796875,-50.90609765625,16],[0.67381045334471,-0.735493605000546,0.0522875687219803,-0.0479024020675531],[0,0,0,0],[8.999999E+09,8.999999E+09,8.999999E+09,8.999999E+09,8.999999E+09,8.999999E+09]];
	LOCAL CONST Robtarget Tr_meulage_bavure_P438 :=[[-123.6238125,-50.78755078125,16],[0.675637238396817,-0.73469627579135,0.0449890485900862,-0.0413725746938977],[0,0,0,0],[8.999999E+09,8.999999E+09,8.999999E+09,8.999999E+09,8.999999E+09,8.999999E+09]];
	LOCAL CONST Robtarget Tr_meulage_bavure_P439 :=[[-129.5069609375,-50.12515234375,16],[0.677409265271052,-0.733888173838118,0.0369228655188245,-0.0340813384033709],[0,0,0,0],[8.999999E+09,8.999999E+09,8.999999E+09,8.999999E+09,8.999999E+09,8.999999E+09]];
	LOCAL CONST Robtarget Tr_meulage_bavure_P440 :=[[-132.771125,-49.92398046875,16],[0.679076860117021,-0.733071427897642,0.0280397377969475,-0.0259744635748024],[0,0,0,0],[8.999999E+09,8.999999E+09,8.999999E+09,8.999999E+09,8.999999E+09,8.999999E+09]];
	LOCAL CONST Robtarget Tr_meulage_bavure_P441 :=[[-134.59365625,-49.8414765625,16],[0.680571808817839,-0.732247971151348,0.018456791550438,-0.0171542599028371],[0,0,0,0],[8.999999E+09,8.999999E+09,8.999999E+09,8.999999E+09,8.999999E+09,8.999999E+09]];
	LOCAL CONST Robtarget Tr_meulage_bavure_P442 :=[[-137.145265625,-49.86151171875,16],[0.681838871122935,-0.731411403481642,0.0084391819880067,-0.00786720345418831],[0,0,0,0],[8.999999E+09,8.999999E+09,8.999999E+09,8.999999E+09,8.999999E+09,8.999999E+09]];
	LOCAL CONST Robtarget Tr_meulage_bavure_P443 :=[[-141.765375,-49.710296875,16],[0.682858343037306,-0.730547498730568,-0.00160645156439322,0.00150158457230694],[0,0,0,0],[8.999999E+09,8.999999E+09,8.999999E+09,8.999999E+09,8.999999E+09,8.999999E+09]];
	LOCAL CONST Robtarget Tr_meulage_bavure_P444 :=[[-143.329625,-49.77455078125,16],[0.683622980266767,-0.729673929214619,-0.0112007535403586,0.0104938551453183],[0,0,0,0],[8.999999E+09,8.999999E+09,8.999999E+09,8.999999E+09,8.999999E+09,8.999999E+09]];
	LOCAL CONST Robtarget Tr_meulage_bavure_P445 :=[[-148.32103125,-50.3141328125,16],[0.684146485042474,-0.728833654698926,-0.0199019150652653,0.0186816637098621],[0,0,0,0],[8.999999E+09,8.999999E+09,8.999999E+09,8.999999E+09,8.999999E+09,8.999999E+09]];
	LOCAL CONST Robtarget Tr_meulage_bavure_P446 :=[[-149.0018125,-50.36703515625,16],[0.684468271768006,-0.728066415598138,-0.0274791377879708,0.0258336293893672],[0,0,0,0],[8.999999E+09,8.999999E+09,8.999999E+09,8.999999E+09,8.999999E+09,8.999999E+09]];
	LOCAL CONST Robtarget Tr_meulage_bavure_P447 :=[[-149.480890625,-50.4411328125,16],[0.684631784042455,-0.727391919141054,-0.0340018215761168,0.0320030057439172],[0,0,0,0],[8.999999E+09,8.999999E+09,8.999999E+09,8.999999E+09,8.999999E+09,8.999999E+09]];
	LOCAL CONST Robtarget Tr_meulage_bavure_P448 :=[[-152.588546875,-50.74232421875,16],[0.684657307917619,-0.726812137517437,-0.0397921866005766,0.037484254799546],[0,0,0,0],[8.999999E+09,8.999999E+09,8.999999E+09,8.999999E+09,8.999999E+09,8.999999E+09]];
	LOCAL CONST Robtarget Tr_meulage_bavure_P449 :=[[-155.93425,-51.2344375,16],[0.684547869571557,-0.726304271328316,-0.045307673376709,0.0427028622983963],[0,0,0,0],[8.999999E+09,8.999999E+09,8.999999E+09,8.999999E+09,8.999999E+09,8.999999E+09]];
	LOCAL CONST Robtarget Tr_meulage_bavure_P450 :=[[-159.2435,-51.64239453125,16],[0.68431475447311,-0.725818883892096,-0.0509336410469018,0.04802112874293],[0,0,0,0],[8.999999E+09,8.999999E+09,8.999999E+09,8.999999E+09,8.999999E+09,8.999999E+09]];
	LOCAL CONST Robtarget Tr_meulage_bavure_P451 :=[[-160.34571875,-51.826109375,16],[0.683946948866958,-0.725326478572325,-0.0569080071676235,0.0536614324972751],[0,0,0,0],[8.999999E+09,8.999999E+09,8.999999E+09,8.999999E+09,8.999999E+09,8.999999E+09]];
	LOCAL CONST Robtarget Tr_meulage_bavure_P452 :=[[-163.50359375,-52.53793359375,16],[0.683439160586235,-0.724800909246756,-0.0633210877913475,0.0597075838832766],[0,0,0,0],[8.999999E+09,8.999999E+09,8.999999E+09,8.999999E+09,8.999999E+09,8.999999E+09]];
	LOCAL CONST Robtarget Tr_meulage_bavure_P453 :=[[-163.591375,-52.55621484375,16],[0.6828158750838,-0.724196225563067,-0.0701747751452285,0.066165009990687],[0,0,0,0],[8.999999E+09,8.999999E+09,8.999999E+09,8.999999E+09,8.999999E+09,8.999999E+09]];
	LOCAL CONST Robtarget Tr_meulage_bavure_P454 :=[[-164.19890625,-52.70726171875,16],[0.682081393576466,-0.723478274853417,-0.0774977450444101,0.0730633825177885],[0,0,0,0],[8.999999E+09,8.999999E+09,8.999999E+09,8.999999E+09,8.999999E+09,8.999999E+09]];
	LOCAL CONST Robtarget Tr_meulage_bavure_P455 :=[[-167.343375,-53.4670859375,16],[0.68123308073897,-0.722619555757437,-0.0852995815382466,0.0804142321558625],[0,0,0,0],[8.999999E+09,8.999999E+09,8.999999E+09,8.999999E+09,8.999999E+09,8.999999E+09]];
	LOCAL CONST Robtarget Tr_meulage_bavure_P456 :=[[-168.093515625,-53.7216640625,16],[0.6802705835487,-0.721609243570014,-0.0935013395899856,0.0881449502098754],[0,0,0,0],[8.999999E+09,8.999999E+09,8.999999E+09,8.999999E+09,8.999999E+09,8.999999E+09]];
	LOCAL CONST Robtarget Tr_meulage_bavure_P457 :=[[-171.1724375,-54.6175703125,16],[0.679225768105469,-0.720441860755123,-0.101907164300553,0.0960771100598499],[0,0,0,0],[8.999999E+09,8.999999E+09,8.999999E+09,8.999999E+09,8.999999E+09,8.999999E+09]];
	LOCAL CONST Robtarget Tr_meulage_bavure_P458 :=[[-172.0349375,-54.839109375,16],[0.678149590660411,-0.719177052709796,-0.110093020915189,0.103812457289749],[0,0,0,0],[8.999999E+09,8.999999E+09,8.999999E+09,8.999999E+09,8.999999E+09,8.999999E+09]];
	LOCAL CONST Robtarget Tr_meulage_bavure_P459 :=[[-175.36403125,-56.0855390625,16],[0.677189205071137,-0.717955933096567,-0.117195438752847,0.110540887467433],[0,0,0,0],[8.999999E+09,8.999999E+09,8.999999E+09,8.999999E+09,8.999999E+09,8.999999E+09]];
	LOCAL CONST Robtarget Tr_meulage_bavure_P460 :=[[-177.356203125,-56.7619609375,16],[0.676599864882265,-0.717032774068392,-0.121869613570241,0.114997482760828],[0,0,0,0],[8.999999E+09,8.999999E+09,8.999999E+09,8.999999E+09,8.999999E+09,8.999999E+09]];
	LOCAL CONST Robtarget Tr_meulage_bavure_P461 :=[[-177.93609375,-57.0348046875,16],[0.676745849817993,-0.716799021565883,-0.122136687679291,0.115311954970183],[0,0,0,0],[8.999999E+09,8.999999E+09,8.999999E+09,8.999999E+09,8.999999E+09,8.999999E+09]];
	LOCAL CONST Robtarget Tr_meulage_bavure_P462 :=[[-179.95846875,-57.90127734375,16],[0.678023751361417,-0.717681357911311,-0.115432129548396,0.10905358574705],[0,0,0,0],[8.999999E+09,8.999999E+09,8.999999E+09,8.999999E+09,8.999999E+09,8.999999E+09]];
	LOCAL CONST Robtarget Tr_meulage_bavure_P463 :=[[-184.21275,-60.053953125,16],[0.680635090594999,-0.719864763536112,-0.0989138766327252,0.0935234766212309],[0,0,0,0],[8.999999E+09,8.999999E+09,8.999999E+09,8.999999E+09,8.999999E+09,8.999999E+09]];
	LOCAL CONST Robtarget Tr_meulage_bavure_P464 :=[[-184.920640625,-60.6799296875,16],[0.68414739288921,-0.722926102139678,-0.0701196541653083,0.0663583434676147],[0,0,0,0],[8.999999E+09,8.999999E+09,8.999999E+09,8.999999E+09,8.999999E+09,8.999999E+09]];
	LOCAL CONST Robtarget Tr_meulage_bavure_P465 :=[[-185.074890625,-60.7686171875,16],[0.687216723794357,-0.72540877583698,-0.0282591369811231,0.0267713214677012],[0,0,0,0],[8.999999E+09,8.999999E+09,8.999999E+09,8.999999E+09,8.999999E+09,8.999999E+09]];
	LOCAL CONST Robtarget Tr_meulage_bavure_P466 :=[[-185.2733125,-60.84550390625,16],[0.687803202537614,-0.725139188448824,0.0240624204820962,-0.022823493933345],[0,0,0,0],[8.999999E+09,8.999999E+09,8.999999E+09,8.999999E+09,8.999999E+09,8.999999E+09]];
	LOCAL CONST Robtarget Tr_meulage_bavure_P467 :=[[-189.130921875,-61.9678203125,16],[0.684474260888735,-0.720609986437375,0.0801379076372037,-0.0761193102115185],[0,0,0,0],[8.999999E+09,8.999999E+09,8.999999E+09,8.999999E+09,8.999999E+09,8.999999E+09]];
	LOCAL CONST Robtarget Tr_meulage_bavure_P468 :=[[-192.087078125,-61.8622890625,16],[0.677761690549222,-0.712392056650159,0.131883604724803,-0.125472559750766],[0,0,0,0],[8.999999E+09,8.999999E+09,8.999999E+09,8.999999E+09,8.999999E+09,8.999999E+09]];
	LOCAL CONST Robtarget Tr_meulage_bavure_P469 :=[[-192.422234375,-61.87291015625,16],[0.669680704265225,-0.702621071014132,0.174107846044042,-0.165945300770136],[0,0,0,0],[8.999999E+09,8.999999E+09,8.999999E+09,8.999999E+09,8.999999E+09,8.999999E+09]];
	LOCAL CONST Robtarget Tr_meulage_bavure_P470 :=[[-192.82253125,-61.5681171875,16],[0.662098384534546,-0.693199887720595,0.205936700494416,-0.196697026541767],[0,0,0,0],[8.999999E+09,8.999999E+09,8.999999E+09,8.999999E+09,8.999999E+09,8.999999E+09]];
	LOCAL CONST Robtarget Tr_meulage_bavure_P471 :=[[-194.415140625,-60.41587890625,16],[0.655812498115986,-0.684945439331905,0.22927756466948,-0.219525649509405],[0,0,0,0],[8.999999E+09,8.999999E+09,8.999999E+09,8.999999E+09,8.999999E+09,8.999999E+09]];
	LOCAL CONST Robtarget Tr_meulage_bavure_P472 :=[[-195.983375,-59.08196875,16],[0.650740291584837,-0.677770298538279,0.24691112080772,-0.237064113161164],[0,0,0,0],[8.999999E+09,8.999999E+09,8.999999E+09,8.999999E+09,8.999999E+09,8.999999E+09]];
	LOCAL CONST Robtarget Tr_meulage_bavure_P473 :=[[-198.624640625,-55.75273046875,16],[0.646450046613984,-0.671170225516012,0.26131429068241,-0.251689703998221],[0,0,0,0],[8.999999E+09,8.999999E+09,8.999999E+09,8.999999E+09,8.999999E+09,8.999999E+09]];
	LOCAL CONST Robtarget Tr_meulage_bavure_P474 :=[[-199.55378125,-54.5555859375,16],[0.642434244032129,-0.664626681012912,0.27430888877872,-0.2651494871155],[0,0,0,0],[8.999999E+09,8.999999E+09,8.999999E+09,8.999999E+09,8.999999E+09,8.999999E+09]];
	LOCAL CONST Robtarget Tr_meulage_bavure_P475 :=[[-200.4540625,-53.62323046875,16],[0.638358403746274,-0.65775675656731,0.286913283781153,-0.27845172857513],[0,0,0,0],[8.999999E+09,8.999999E+09,8.999999E+09,8.999999E+09,8.999999E+09,8.999999E+09]];
	LOCAL CONST Robtarget Tr_meulage_bavure_P476 :=[[-202.516734375,-51.28213671875,16],[0.634071841159138,-0.650411982924208,0.299471814695801,-0.291948257265675],[0,0,0,0],[8.999999E+09,8.999999E+09,8.999999E+09,8.999999E+09,8.999999E+09,8.999999E+09]];
	LOCAL CONST Robtarget Tr_meulage_bavure_P477 :=[[-204.09425,-49.3264765625,16],[0.629655243905703,-0.642696245944215,0.311753086074583,-0.305427278732985],[0,0,0,0],[8.999999E+09,8.999999E+09,8.999999E+09,8.999999E+09,8.999999E+09,8.999999E+09]];
	LOCAL CONST Robtarget Tr_meulage_bavure_P478 :=[[-205.974359375,-46.5244140625,16],[0.625464154096542,-0.634992237105909,0.323022691870682,-0.318175723920207],[0,0,0,0],[8.999999E+09,8.999999E+09,8.999999E+09,8.999999E+09,8.999999E+09,8.999999E+09]];
	LOCAL CONST Robtarget Tr_meulage_bavure_P479 :=[[-208.261046875,-42.804109375,16],[0.62197513707743,-0.627820617035987,0.332442955570272,-0.329347662772588],[0,0,0,0],[8.999999E+09,8.999999E+09,8.999999E+09,8.999999E+09,8.999999E+09,8.999999E+09]];
	LOCAL CONST Robtarget Tr_meulage_bavure_P480 :=[[-208.56609375,-42.378875,16],[0.61960816252237,-0.621606676412682,0.339433738687335,-0.33834243277421],[0,0,0,0],[8.999999E+09,8.999999E+09,8.999999E+09,8.999999E+09,8.999999E+09,8.999999E+09]];
	LOCAL CONST Robtarget Tr_meulage_bavure_P481 :=[[-210.421875,-39.5615546875,16],[0.618452186711343,-0.616499019158342,0.344016552882489,-0.345106452376089],[0,0,0,0],[8.999999E+09,8.999999E+09,8.999999E+09,8.999999E+09,8.999999E+09,8.999999E+09]];
	LOCAL CONST Robtarget Tr_meulage_bavure_P482 :=[[-212.59271875,-35.97863671875,16],[0.618178619804139,-0.612240725736773,0.346894069264997,-0.350258465244069],[0,0,0,0],[8.999999E+09,8.999999E+09,8.999999E+09,8.999999E+09,8.999999E+09,8.999999E+09]];
	LOCAL CONST Robtarget Tr_meulage_bavure_P483 :=[[-215.5064375,-31.36932421875,16],[0.618212329859709,-0.608258572608231,0.349150787118479,-0.354864413420921],[0,0,0,0],[8.999999E+09,8.999999E+09,8.999999E+09,8.999999E+09,8.999999E+09,8.999999E+09]];
	LOCAL CONST Robtarget Tr_meulage_bavure_P484 :=[[-215.820515625,-30.886078125,16],[0.617876211426908,-0.604025228883112,0.351879783538558,-0.35994878547134],[0,0,0,0],[8.999999E+09,8.999999E+09,8.999999E+09,8.999999E+09,8.999999E+09,8.999999E+09]];
	LOCAL CONST Robtarget Tr_meulage_bavure_P485 :=[[-217.2355,-28.7861015625,16],[0.616737718495692,-0.599207918130712,0.355719366610983,-0.366125920486473],[0,0,0,0],[8.999999E+09,8.999999E+09,8.999999E+09,8.999999E+09,8.999999E+09,8.999999E+09]];
	LOCAL CONST Robtarget Tr_meulage_bavure_P486 :=[[-218.319125,-27.22653125,16],[0.614709081978266,-0.593813388514203,0.360694532504914,-0.373387008847093],[0,0,0,0],[8.999999E+09,8.999999E+09,8.999999E+09,8.999999E+09,8.999999E+09,8.999999E+09]];
	LOCAL CONST Robtarget Tr_meulage_bavure_P487 :=[[-219.760609375,-24.640625,16],[0.612027132244768,-0.588168674285347,0.36631497143641,-0.381174161882996],[0,0,0,0],[8.999999E+09,8.999999E+09,8.999999E+09,8.999999E+09,8.999999E+09,8.999999E+09]];
	LOCAL CONST Robtarget Tr_meulage_bavure_P488 :=[[-220.511671875,-23.34393359375,16],[0.609132958520891,-0.582764428746032,0.371851164906505,-0.388676434312106],[0,0,0,0],[8.999999E+09,8.999999E+09,8.999999E+09,8.999999E+09,8.999999E+09,8.999999E+09]];
	LOCAL CONST Robtarget Tr_meulage_bavure_P489 :=[[-220.848140625,-22.7561640625,16],[0.606445141732903,-0.578103163045802,0.376674953315704,-0.395141749869094],[0,0,0,0],[8.999999E+09,8.999999E+09,8.999999E+09,8.999999E+09,8.999999E+09,8.999999E+09]];
	LOCAL CONST Robtarget Tr_meulage_bavure_P490 :=[[-221.635609375,-20.804259765625,16],[0.604333048493108,-0.574551079630144,0.380321341855554,-0.400035373840933],[0,0,0,0],[8.999999E+09,8.999999E+09,8.999999E+09,8.999999E+09,8.999999E+09,8.999999E+09]];
	LOCAL CONST Robtarget Tr_meulage_bavure_P491 :=[[-222.035890625,-19.727814453125,16],[0.603001202057322,-0.572350075401805,0.382563518190902,-0.403050984435433],[0,0,0,0],[8.999999E+09,8.999999E+09,8.999999E+09,8.999999E+09,8.999999E+09,8.999999E+09]];
	LOCAL CONST Robtarget Tr_meulage_bavure_P492 :=[[-222.368765625,-16.604248046875,16],[0.60254414781958,-0.571606822841799,0.383321330967731,-0.404067998280249],[0,0,0,0],[8.999999E+09,8.999999E+09,8.999999E+09,8.999999E+09,8.999999E+09,8.999999E+09]];
	LOCAL CONST Robtarget Tr_meulage_bavure_degg1 :=[[-231.607486613361,-20.3948573079714,15.4733920538834],[0.60254414781958,-0.571606822841799,0.383321330967731,-0.404067998280249],[0,0,0,0],[8.999999E+09,8.999999E+09,8.999999E+09,8.999999E+09,8.999999E+09,8.999999E+09]];
	LOCAL CONST Robtarget Tr_meulage_bavure_degg2 :=[[-407.143185392215,-92.4164332688022,5.46784107766739],[0.60254414781958,-0.571606822841799,0.383321330967731,-0.404067998280249],[0,0,0,0],[8.999999E+09,8.999999E+09,8.999999E+09,8.999999E+09,8.999999E+09,8.999999E+09]];
	LOCAL PROC Tr_pick()
		!!Programme Tr_pick - 28/02/2023 14:23:08;
		 CONST Robtarget Ppick :=[[-8.56999969482422,13.3900003433228,624.75],[0.00458215070835504,0.917000799761137,-0.398780045054065,0.00793806015339623],[0,0,0,0],[8.999999E+09,8.999999E+09,8.999999E+09,8.999999E+09,8.999999E+09,8.999999E+09]];
		 VAR Pose Ref :=[[0,0,0],[1,0,0,0]];
		LocalisationPieceTable 61 \model:=0;
		MoveJ Reltool(Ppick,0,0,-200),V1000,Z0,Tool_Prehenseur \Wobj:=Wobj_vision;
		MoveL Reltool(Ppick,0,0,-100),V500,Z0,Tool_Prehenseur \Wobj:=Wobj_vision;
		MoveL Reltool(Ppick,0,0,-10),V200,Z0,Tool_Prehenseur \Wobj:=Wobj_vision;
		MoveL Ppick,V100,Fine,Tool_Prehenseur \Wobj:=Wobj_vision;
		Gripper_Close;
		MoveL Reltool(Ppick,0,0,-200),V500,Z0,Tool_Prehenseur \Wobj:=Wobj_vision;
		LocalisationPiecePrehenseur 61 \model:=0,Ref;
	ENDPROC
	LOCAL PROC Tr_Cut()
		!!Programme Tr_Cut - 28/02/2023 14:23:08;
		confJ \off;
		confL \off;
		Tool := ToolOffset(Tool_M2_D490_S180);
		MoveAbsJ [[0,-40,40,0,90,0],[8.999999E+09,8.999999E+09,8.999999E+09,8.999999E+09,8.999999E+09,8.999999E+09]] ,V1000,Z0,Tool_M2_D490_S180 \Wobj:=Wobj_Part_0;
		Movej Reltool(Coupe_0,-200,0,-47.1993359375),V1000,Z0,Tool_M2_D490_S180 \Wobj:=Wobj_Part_0;
		MoveL Reltool(Coupe_0,0,0,-47.1993359375),V500,Z0,Tool_M2_D490_S180 \Wobj:=Wobj_Part_0;
		MoveL Reltool(Coupe_0,0,0,-37.1993359375),vitesse_Tronconnage,Z0,Tool_M2_D490_S180 \Wobj:=Wobj_Part_0;
		MoveL Coupe_0,vitesse_Tronconnage,Fine,Tool_M2_D490_S180 \Wobj:=Wobj_Part_0;
		MoveL Reltool(Coupe_0,0,0,37.1993359375),vitesse_Tronconnage,Z0,Tool_M2_D490_S180 \Wobj:=Wobj_Part_0;
		MoveL Reltool(Coupe_0,-200,0,37.1993359375),V500,Z0,Tool_M2_D490_S180 \Wobj:=Wobj_Part_0;
		MoveAbsJ [[0,-40,40,0,90,0],[8.999999E+09,8.999999E+09,8.999999E+09,8.999999E+09,8.999999E+09,8.999999E+09]] ,V1000,Z0,Tool_M2_D490_S180 \Wobj:=Wobj_Part_0;
		Movej Reltool(Coupe_1,-200,0,-43.5283515625),V1000,Z0,Tool_M2_D490_S180 \Wobj:=Wobj_Part_0;
		MoveL Reltool(Coupe_1,0,0,-43.5283515625),V500,Z0,Tool_M2_D490_S180 \Wobj:=Wobj_Part_0;
		MoveL Reltool(Coupe_1,0,0,-33.5283515625),vitesse_Tronconnage,Z0,Tool_M2_D490_S180 \Wobj:=Wobj_Part_0;
		MoveL Coupe_1,vitesse_Tronconnage,Fine,Tool_M2_D490_S180 \Wobj:=Wobj_Part_0;
		MoveL Reltool(Coupe_1,0,0,33.5283515625),vitesse_Tronconnage,Z0,Tool_M2_D490_S180 \Wobj:=Wobj_Part_0;
		MoveL Reltool(Coupe_1,-200,0,33.5283515625),V500,Z0,Tool_M2_D490_S180 \Wobj:=Wobj_Part_0;
	ENDPROC
	LOCAL PROC Tr_meulage_motif_1()
		!!Programme Tr_meulage_motif_1 - 28/02/2023 14:23:08;
		 CONST Speeddata vitesse_Meulage :=[50, 500, 0, 0];
		confJ \off;
		confL \off;
		Tool := ToolOffset(Tool_M1_D500_S270);
		MoveAbsJ [[0,-40,40,0,90,0],[8.999999E+09,8.999999E+09,8.999999E+09,8.999999E+09,8.999999E+09,8.999999E+09]] ,V1000,Z0,Tool_M1_D500_S270 \Wobj:=Wobj_Part_0;
		MoveJ Tr_meulage_motif_1_App1,V2000,Z100,Tool,\Wobj:=Wobj_Part_0;
		MoveJ Tr_meulage_motif_1_App2,V500,Z0,Tool,\Wobj:=Wobj_Part_0;
		MoveL Tr_meulage_motif_1_P0,[12.5,500,0,0],z0,Tool \wobj:=Wobj_Part_0;
		MoveL Tr_meulage_motif_1_P1,[12.5,500,0,0],z0,Tool \wobj:=Wobj_Part_0;
		MoveL Tr_meulage_motif_1_P2,[12.5,500,0,0],z0,Tool \wobj:=Wobj_Part_0;
		MoveL Tr_meulage_motif_1_P3,[12.5,500,0,0],z0,Tool \wobj:=Wobj_Part_0;
		MoveL Tr_meulage_motif_1_P4,[12.5,500,0,0],z0,Tool \wobj:=Wobj_Part_0;
		MoveL Tr_meulage_motif_1_P5,[12.5,500,0,0],z0,Tool \wobj:=Wobj_Part_0;
		MoveL Tr_meulage_motif_1_P6,[12.5,500,0,0],z0,Tool \wobj:=Wobj_Part_0;
		MoveL Tr_meulage_motif_1_P7,[12.5,500,0,0],z0,Tool \wobj:=Wobj_Part_0;
		MoveL Tr_meulage_motif_1_P8,[12.5,500,0,0],z0,Tool \wobj:=Wobj_Part_0;
		MoveL Tr_meulage_motif_1_P9,[12.5,500,0,0],z0,Tool \wobj:=Wobj_Part_0;
		MoveL Tr_meulage_motif_1_P10,[12.5,500,0,0],z0,Tool \wobj:=Wobj_Part_0;
		MoveL Tr_meulage_motif_1_P11,[12.5,500,0,0],z0,Tool \wobj:=Wobj_Part_0;
		MoveL Tr_meulage_motif_1_P12,[12.5,500,0,0],z0,Tool \wobj:=Wobj_Part_0;
		MoveL Tr_meulage_motif_1_P13,[12.5,500,0,0],z0,Tool \wobj:=Wobj_Part_0;
		MoveL Tr_meulage_motif_1_P14,[12.5,500,0,0],z0,Tool \wobj:=Wobj_Part_0;
		MoveL Tr_meulage_motif_1_P15,[12.5,500,0,0],z0,Tool \wobj:=Wobj_Part_0;
		MoveL Tr_meulage_motif_1_P16,[12.5,500,0,0],z0,Tool \wobj:=Wobj_Part_0;
		MoveL Tr_meulage_motif_1_P17,[12.5,500,0,0],z0,Tool \wobj:=Wobj_Part_0;
		MoveL Tr_meulage_motif_1_P18,[12.5,500,0,0],z0,Tool \wobj:=Wobj_Part_0;
		MoveL Tr_meulage_motif_1_P19,[12.5,500,0,0],z0,Tool \wobj:=Wobj_Part_0;
		MoveL Tr_meulage_motif_1_P20,[12.5,500,0,0],z0,Tool \wobj:=Wobj_Part_0;
		MoveL Tr_meulage_motif_1_P21,[12.5,500,0,0],z0,Tool \wobj:=Wobj_Part_0;
		MoveL Tr_meulage_motif_1_P22,[12.5,500,0,0],z0,Tool \wobj:=Wobj_Part_0;
		MoveL Tr_meulage_motif_1_P23,[12.5,500,0,0],z0,Tool \wobj:=Wobj_Part_0;
		MoveL Tr_meulage_motif_1_P24,[12.5,500,0,0],z0,Tool \wobj:=Wobj_Part_0;
		MoveL Tr_meulage_motif_1_P25,[12.5,500,0,0],z0,Tool \wobj:=Wobj_Part_0;
		MoveL Tr_meulage_motif_1_P26,[12.5,500,0,0],z0,Tool \wobj:=Wobj_Part_0;
		MoveL Tr_meulage_motif_1_P27,[12.5,500,0,0],z0,Tool \wobj:=Wobj_Part_0;
		MoveL Tr_meulage_motif_1_P28,[12.5,500,0,0],z0,Tool \wobj:=Wobj_Part_0;
		MoveL Tr_meulage_motif_1_P29,[12.5,500,0,0],z0,Tool \wobj:=Wobj_Part_0;
		MoveL Tr_meulage_motif_1_P30,[12.5,500,0,0],z0,Tool \wobj:=Wobj_Part_0;
		MoveL Tr_meulage_motif_1_P31,[12.5,500,0,0],z0,Tool \wobj:=Wobj_Part_0;
		MoveL Tr_meulage_motif_1_P32,[12.5,500,0,0],z0,Tool \wobj:=Wobj_Part_0;
		MoveL Tr_meulage_motif_1_P33,[12.5,500,0,0],z0,Tool \wobj:=Wobj_Part_0;
		MoveL Tr_meulage_motif_1_P34,[12.5,500,0,0],z0,Tool \wobj:=Wobj_Part_0;
		MoveL Tr_meulage_motif_1_P35,[12.5,500,0,0],z0,Tool \wobj:=Wobj_Part_0;
		MoveL Tr_meulage_motif_1_P36,[12.5,500,0,0],z0,Tool \wobj:=Wobj_Part_0;
		MoveL Tr_meulage_motif_1_P37,[12.5,500,0,0],z0,Tool \wobj:=Wobj_Part_0;
		MoveL Tr_meulage_motif_1_P38,[12.5,500,0,0],z0,Tool \wobj:=Wobj_Part_0;
		MoveL Tr_meulage_motif_1_P39,[12.5,500,0,0],z0,Tool \wobj:=Wobj_Part_0;
		MoveL Tr_meulage_motif_1_P40,[12.5,500,0,0],z0,Tool \wobj:=Wobj_Part_0;
		MoveL Tr_meulage_motif_1_P41,[12.5,500,0,0],z0,Tool \wobj:=Wobj_Part_0;
		MoveL Tr_meulage_motif_1_P42,[12.5,500,0,0],z0,Tool \wobj:=Wobj_Part_0;
		MoveL Tr_meulage_motif_1_P43,[12.5,500,0,0],z0,Tool \wobj:=Wobj_Part_0;
		MoveL Tr_meulage_motif_1_P44,[12.5,500,0,0],z0,Tool \wobj:=Wobj_Part_0;
		MoveL Tr_meulage_motif_1_P45,[12.5,500,0,0],z0,Tool \wobj:=Wobj_Part_0;
		MoveL Tr_meulage_motif_1_P46,[12.5,500,0,0],z0,Tool \wobj:=Wobj_Part_0;
		MoveL Tr_meulage_motif_1_P47,[12.5,500,0,0],z0,Tool \wobj:=Wobj_Part_0;
		MoveL Tr_meulage_motif_1_P48,[12.5,500,0,0],z0,Tool \wobj:=Wobj_Part_0;
		MoveL Tr_meulage_motif_1_P49,[12.5,500,0,0],z0,Tool \wobj:=Wobj_Part_0;
		MoveL Tr_meulage_motif_1_P50,[12.5,500,0,0],z0,Tool \wobj:=Wobj_Part_0;
		MoveL Tr_meulage_motif_1_P51,[12.5,500,0,0],z0,Tool \wobj:=Wobj_Part_0;
		MoveL Tr_meulage_motif_1_P52,[12.5,500,0,0],z0,Tool \wobj:=Wobj_Part_0;
		MoveL Tr_meulage_motif_1_P53,[12.5,500,0,0],z0,Tool \wobj:=Wobj_Part_0;
		MoveL Tr_meulage_motif_1_P54,[12.5,500,0,0],z0,Tool \wobj:=Wobj_Part_0;
		MoveL Tr_meulage_motif_1_P55,[12.5,500,0,0],z0,Tool \wobj:=Wobj_Part_0;
		MoveL Tr_meulage_motif_1_P56,[12.5,500,0,0],z0,Tool \wobj:=Wobj_Part_0;
		MoveL Tr_meulage_motif_1_P57,[12.5,500,0,0],z0,Tool \wobj:=Wobj_Part_0;
		MoveL Tr_meulage_motif_1_P58,[12.5,500,0,0],z0,Tool \wobj:=Wobj_Part_0;
		MoveL Tr_meulage_motif_1_P59,[12.5,500,0,0],z0,Tool \wobj:=Wobj_Part_0;
		MoveL Tr_meulage_motif_1_P60,[12.5,500,0,0],z0,Tool \wobj:=Wobj_Part_0;
		MoveL Tr_meulage_motif_1_P61,[12.5,500,0,0],z0,Tool \wobj:=Wobj_Part_0;
		MoveL Tr_meulage_motif_1_P62,[12.5,500,0,0],z0,Tool \wobj:=Wobj_Part_0;
		MoveL Tr_meulage_motif_1_P63,[12.5,500,0,0],z0,Tool \wobj:=Wobj_Part_0;
		MoveL Tr_meulage_motif_1_P64,[12.5,500,0,0],z0,Tool \wobj:=Wobj_Part_0;
		MoveL Tr_meulage_motif_1_P65,[12.5,500,0,0],z0,Tool \wobj:=Wobj_Part_0;
		MoveL Tr_meulage_motif_1_P66,[12.5,500,0,0],z0,Tool \wobj:=Wobj_Part_0;
		MoveL Tr_meulage_motif_1_P67,[12.5,500,0,0],z0,Tool \wobj:=Wobj_Part_0;
		MoveL Tr_meulage_motif_1_P68,[12.5,500,0,0],z0,Tool \wobj:=Wobj_Part_0;
		MoveL Tr_meulage_motif_1_P69,[12.5,500,0,0],z0,Tool \wobj:=Wobj_Part_0;
		MoveL Tr_meulage_motif_1_P70,[12.5,500,0,0],z0,Tool \wobj:=Wobj_Part_0;
		MoveL Tr_meulage_motif_1_P71,[12.5,500,0,0],z0,Tool \wobj:=Wobj_Part_0;
		MoveL Tr_meulage_motif_1_P72,[12.5,500,0,0],z0,Tool \wobj:=Wobj_Part_0;
		MoveL Tr_meulage_motif_1_P73,[12.5,500,0,0],z0,Tool \wobj:=Wobj_Part_0;
		MoveL Tr_meulage_motif_1_P74,[12.5,500,0,0],z0,Tool \wobj:=Wobj_Part_0;
		MoveL Tr_meulage_motif_1_P75,[12.5,500,0,0],z0,Tool \wobj:=Wobj_Part_0;
		MoveL Tr_meulage_motif_1_P76,[12.5,500,0,0],z0,Tool \wobj:=Wobj_Part_0;
